// TIA Portal project "Hgu_controller" (V17)

(* hardware
DEVICE "S7-1500/ET200MP station_1"  S7-1500 station
   slot 0: "Rail_0"  Rack  6ES7 590-1***0-0AA0
   slot 1: "HGU_Controller"  CPU 1511-1 PN  6ES7 511-1AK02-0AB0  V2.9
      slot 3: "CPU display_1"  6ES7591-1AA00-0AA0
      slot 32768: "PROFINET interface_1"  X1
         slot 32769: "Port_1"  X1 P1
         slot 32770: "Port_2"  X1 P2
      slot 34817: "Virtual CP interface port_1"  Virtual CP interface port  Virtual CP interface port
DEVICE "ET 200SP station_1"  ET 200SP-Station
   slot 0: "Rack_0"  Rack  6ES5 710-8MAx1
   slot 0: "HPU"  IM 155-6 PN ST  6ES7 155-6AU01-0BN0  V4.2
   slot 1: "DI 16x24VDC ST_1"  DI 16x24VDC ST  6ES7 131-6BH01-0BA0  V0.0
      slot 1: "DI 16x24VDC ST_1"  DI 16x24VDC ST
   slot 2: "DI 16x24VDC ST_2"  DI 16x24VDC ST  6ES7 131-6BH01-0BA0  V0.0
      slot 1: "DI 16x24VDC ST_2"  DI 16x24VDC ST
   slot 3: "DQ 16x24VDC/0.5A ST_1"  DQ 16x24VDC/0.5A ST  6ES7 132-6BH01-0BA0  V0.0
      slot 1: "DQ 16x24VDC/0.5A ST_1"  DQ 16x24VDC/0.5A ST
   slot 4: "AI 4xU/I 2-wire ST_1"  AI 4xU/I 2-wire ST  6ES7 134-6HD01-0BA1  V2.0
      slot 1: "AI 4xU/I 2-wire ST_1"  AI 4xU/I 2-wire ST
   slot 5: "AI 4xU/I 2-wire ST_2"  AI 4xU/I 2-wire ST  6ES7 134-6HD01-0BA1  V2.0
      slot 1: "AI 4xU/I 2-wire ST_2"  AI 4xU/I 2-wire ST
   slot 6: "AI 4xU/I 2-wire ST_3"  AI 4xU/I 2-wire ST  6ES7 134-6HD01-0BA1  V2.0
      slot 1: "AI 4xU/I 2-wire ST_3"  AI 4xU/I 2-wire ST
   slot 7: "AI 4xU/I 2-wire ST_4"  AI 4xU/I 2-wire ST  6ES7 134-6HD01-0BA1  V2.0
      slot 1: "AI 4xU/I 2-wire ST_4"  AI 4xU/I 2-wire ST
   slot 8: "AI 4xU/I 2-wire ST_5"  AI 4xU/I 2-wire ST  6ES7 134-6HD01-0BA1  V2.0
      slot 1: "AI 4xU/I 2-wire ST_5"  AI 4xU/I 2-wire ST
   slot 9: "CM PtP_1"  CM PtP  6ES7 137-6AA00-0BA0  V1.0
      slot 1: "CM PtP_1"  CM PtP Sub
   slot 10: "Server module_1"  Server module  6ES7 193-6PA00-0AA0  V1.1
      slot 1: "Server module_1"  Server module
   slot 127: "BA 2xRJ45"  BA 2xRJ45  6ES7 193-6AR00-0AA0  V0.0
      slot 1: "Port_1"  X1 P1 R  6ES7 193-6AR00-0AA0  V0.0
      slot 2: "Port_2"  X1 P2 R  6ES7 193-6AR00-0AA0  V0.0
DEVICE "SINAMICS G_1"  Sinamics.Device
   slot 0: "	_0"  Rail  SinamicsG120CRackP
   slot 0: "Drive_1"  G120C PN  6SL3210-1KE31-7AF1  4.7.13
      slot 1: "PROFINET interface"  MDD-SinamicsG120-P
      slot 3: "PM G120C"  PM G120C  6SL3210-1KE31-7AF1  -
DEVICE "SINAMICS G_2"  Sinamics.Device
   slot 0: "	_0"  Rail  SinamicsG120CRackP
   slot 0: "Drive_2"  G120C PN  6SL3210-1KE31-7AF1  4.7.13
      slot 1: "PROFINET interface"  MDD-SinamicsG120-P
      slot 3: "PM G120C"  PM G120C  6SL3210-1KE31-7AF1  -
DEVICE "SINAMICS G_3"  Sinamics.Device
   slot 0: "	_0"  Rail  SinamicsG120CRackP
   slot 0: "Drive_3"  G120C PN  6SL3210-1KE31-7AF1  4.7.13
      slot 1: "PROFINET interface"  MDD-SinamicsG120-P
      slot 3: "PM G120C"  PM G120C  6SL3210-1KE31-7AF1  -
DEVICE "SINAMICS G_4"  Sinamics.Device
   slot 0: "	_0"  Rail  SinamicsG120CRackP
   slot 0: "Drive_4"  G120C PN  6SL3210-1KE31-7AF1  4.7.13
      slot 1: "PROFINET interface"  MDD-SinamicsG120-P
      slot 3: "PM G120C"  PM G120C  6SL3210-1KE31-7AF1  -
DEVICE "SINAMICS G_6"  Sinamics.Device
   slot 0: "	_0"  Rail  SinamicsG120CRackP
   slot 0: "Drive_6"  G120C PN  6SL3210-1KE31-7AF1  4.7.13
      slot 1: "PROFINET interface"  MDD-SinamicsG120-P
      slot 3: "PM G120C"  PM G120C  6SL3210-1KE31-7AF1  -
DEVICE "ET 200SP station_2"  ET 200SP-Station
   slot 0: "Rack_0"  Rack  6ES5 710-8MAx1
   slot 0: "Main Cabinet"  IM 155-6 PN ST  6ES7 155-6AU01-0BN0  V4.2
   slot 1: "DI 16x24VDC ST_1"  DI 16x24VDC ST  6ES7 131-6BH01-0BA0  V0.0
      slot 1: "DI 16x24VDC ST_1"  DI 16x24VDC ST
   slot 2: "DI 16x24VDC ST_2"  DI 16x24VDC ST  6ES7 131-6BH01-0BA0  V0.0
      slot 1: "DI 16x24VDC ST_2"  DI 16x24VDC ST
   slot 3: "DQ 16x24VDC/0.5A ST_1"  DQ 16x24VDC/0.5A ST  6ES7 132-6BH01-0BA0  V0.0
      slot 1: "DQ 16x24VDC/0.5A ST_1"  DQ 16x24VDC/0.5A ST
   slot 4: "Server module_01"  Server module  6ES7 193-6PA00-0AA0  V1.1
      slot 1: "Server module_01"  Server module
   slot 127: "BA 2xRJ45"  BA 2xRJ45  6ES7 193-6AR00-0AA0  V0.0
      slot 1: "Port_1"  X1 P1 R  6ES7 193-6AR00-0AA0  V0.0
      slot 2: "Port_2"  X1 P2 R  6ES7 193-6AR00-0AA0  V0.0
*)

// ===== PLC "HGU_Controller"  CPU 1511-1 PN =====

VAR_GLOBAL   // PLC tag table "Default tag table"
   "Motor1MpcbFault" AT %I44.0 : Bool;   // Motor1 Mks Termik Hata
   "Motor2MpcbFault" AT %I44.1 : Bool;   // Motor 2 Mks Termik Hata
   "Motor3MpcbFault" AT %I44.2 : Bool;   // Motor 3 Mks Termik Hata
   "Motor4MpcbFault" AT %I44.3 : Bool;   // Motor 4 Mks Termik Hata
   "Motor5MpcbFault" AT %I44.4 : Bool;   // Motor 5 Mks Termik Hata
   "Motor6MpcbFault" AT %I44.5 : Bool;   // Motor 6 Mks Termik Hata
   "CoilTubeSoftStarterRunning" AT %I44.6 : Bool;   // Coiltube Yumuşak Yol Verici Çalışıyor
   "CoilTubeSoftStarterContactor" AT %I44.7 : Bool;   // Coiltube Yumuşak Yol Verici Kontaktör Devrede
   "CoilTubeMpcbFault" AT %I45.0 : Bool;   // Coiltube Mks Termik Hata
   "CircSoftStarterRunning" AT %I45.1 : Bool;   // Sirkülasyon Yumuşak Yol Verici Çalışıyor
   "CircSoftStarterContactor" AT %I45.2 : Bool;   // Sirkülasyon Yumuşak Yol Verici Kontaktör Devrede
   "CircMpcbFault" AT %I45.3 : Bool;   // Sirkülasyon Mks Termik Hata
   "ParticleContactorEngaged" AT %I45.4 : Bool;   // Particle Measurement Contactor Engaged
   "ParticleMpcbFault" AT %I45.5 : Bool;   // Particle Measurement Mks Termik Hata
   "PhaseProtectionOk" AT %I45.6 : Bool;   // Faz Koruma Rölesi Ok
   "SafetyRelayOk" AT %I45.7 : Bool;   // Emniyet Rölesi Ok
   "MainSwitchAlarm" AT %I46.0 : Bool;   // Ana Şalter Alarm Kontağı
   "ToroidalLeakageFuse" AT %I46.1 : Bool;   // Toroidal Kaçak Akım Rölesi Sigorta Bilgisi
   "ToroidalLeakageAlarm" AT %I46.2 : Bool;   // Toroidal Kaçak Akım Rölesi Alarm
   "EmergencyStopPlcStatus" AT %I46.3 : Bool;   // Acil Stop Butonu Plc Durum
   "EmergencyStopGpStatus" AT %I46.4 : Bool;   // Acil Stop Butonu Gb Durum
   "ControlPhaseFuse220Vac" AT %I46.5 : Bool;   // 220Vac Kumanda Faz Sigortası Bilgisi
   "EnergyAnalyzerLeakageRelay" AT %I46.6 : Bool;   // Enerji Analizörü Besleme Kaçak Akım Rölesi
   "SignalTowerGreen" AT %Q20.0 : Bool;   // Işık Kulesi Yeşil
   "SignalTowerYellow" AT %Q20.1 : Bool;   // Işık Kulesi Sarı
   "SignalTowerRed" AT %Q20.2 : Bool;   // Işık Kulesi Kırmızı
   "SignalTowerBuzzer" AT %Q20.3 : Bool;   // Işık Kulesi Buzzer
   "ParticleMotorCmd" AT %Q20.4 : Bool;   // Particle Measurement Motor 1/0 Komutu
   "CircContactorCmd" AT %Q20.5 : Bool;   // Sirkülasyon Kontaktör Komutu
   "CircSoftStarterCmd" AT %Q20.6 : Bool;   // Sirkülasyon Yumuşak Yol Verici Komutu
   "CoilTubeContactorCmd" AT %Q20.7 : Bool;   // Coiltube Kontaktör Komutu
   "CoilTubeSoftStarterCmd" AT %Q21.0 : Bool;   // Coiltube Yumuşak Yol Verici Komutu
   "EmergencyStopUnit1" AT %I0.0 : Bool;   // Acil Durdurma Butonu Ünite 1
   "EmergencyStopUnit2" AT %I0.1 : Bool;   // Acil Durdurma Butonu Ünite 2
   "EmergencyStopUnit3" AT %I0.2 : Bool;   // Acil Durdurma Butonu Ünite 3
   "EmergencyStopUnit4" AT %I0.3 : Bool;   // Acil Durdurma Butonu Ünite 4
   "Motor1FilterWarning" AT %I0.4 : Bool;   // Motor 1 Basınç Hattı Filtresi Uyarı
   "Motor1FilterError" AT %I0.5 : Bool;   // Motor 1 Basınç Hattı Filtresi Hata
   "Motor2FilterWarning" AT %I0.6 : Bool;   // Motor 2 Basınç Hattı Filtresi Uyarı
   "Motor2FilterError" AT %I0.7 : Bool;   // Motor 2 Basınç Hattı Filtresi Hata
   "Motor3FilterWarning" AT %I1.0 : Bool;   // Motor 3 Basınç Hattı Filtresi Uyarı
   "Motor3FilterError" AT %I1.1 : Bool;   // Motor 3 Basınç Hattı Filtresi Hata
   "Motor4FilterWarning" AT %I1.2 : Bool;   // Motor 4 Basınç Hattı Filtresi Uyarı
   "Motor4FilterError" AT %I1.3 : Bool;   // Motor 4 Basınç Hattı Filtresi Hata
   "Motor5FilterWarning" AT %I1.4 : Bool;   // Motor 5 Basınç Hattı Filtresi Uyarı
   "Motor5FilterError" AT %I1.5 : Bool;   // Motor 5 Basınç Hattı Filtresi Hata
   "Motor6FilterWarning" AT %I1.6 : Bool;   // Motor 6 Basınç Hattı Filtresi Uyarı
   "Motor6FilterError" AT %I1.7 : Bool;   // Motor 6 Basınç Hattı Filtresi Hata
   "CoilTubeFilterWarning" AT %I2.0 : Bool;   // Coiltube Basınç Hattı Filtresi Uyarı
   "CoilTubeFilterError" AT %I2.1 : Bool;   // Coiltube Basınç Hattı Filtresi Hata
   "TankMinLevelSwitch" AT %I2.2 : Bool;   // Tank Min Seviye Şalteri
   "TankMaxLevelSwitch" AT %I2.3 : Bool;   // Tank Max Seviye Şalteri
   "Motor1CompensatedValve" AT %I2.4 : Bool;   // Motor 1 Kompansatörlü Vana
   "Motor2CompensatedValve" AT %I2.5 : Bool;   // Motor 2 Kompansatörlü Vana
   "Motor3CompensatedValve" AT %I2.6 : Bool;   // Motor 3 Kompansatörlü Vana
   "Motor4CompensatedValve" AT %I2.7 : Bool;   // Motor 4 Kompansatörlü Vana
   "Motor5CompensatedValve" AT %I3.0 : Bool;   // Motor 5 Kompansatörlü Vana
   "Motor6CompensatedValve" AT %I3.1 : Bool;   // Motor 6 Kompansatörlü Vana
   "ChillerWaterFlowSensor" AT %I3.2 : Bool;   // Chiller Su Akış Sensoru
   "TemperatureSensor" AT %IW4 : Int;   // Sıcaklık Sensörü
   "ContinuousLevelSensor" AT %IW6 : Int;   // Sürekli Seviye Sensörü
   "AquaSensor" AT %IW8 : Int;   // Aqua Sensörü
   "PressureTransmitter1" AT %IW10 : Int;   // Basınç Transmitteri 1
   "PressureTransmitter2" AT %IW12 : Int;   // Basınç Transmitteri 2
   "PressureTransmitter3" AT %IW14 : Int;   // Basınç Transmitteri 3
   "PressureTransmitter4" AT %IW16 : Int;   // Basınç Transmitteri 4
   "PressureTransmitter5" AT %IW18 : Int;   // Basınç Transmitteri 5
   "PressureTransmitter6" AT %IW20 : Int;   // Basınç Transmitteri 6
   "CoilTubePressureTransmitter" AT %IW22 : Int;   // Coiltube Basınç Transmitteri
   "Hsm1PressureTransmitter" AT %IW24 : Int;   // Hsm1 Basınç Transmitteri
   "Hsm2PressureTransmitter" AT %IW26 : Int;   // Hsm2 Basınç Transmitteri
   "Hsm3PressureTransmitter" AT %IW28 : Int;   // Hsm3 Basınç Transmitteri
   "Hsm4PressureTransmitter" AT %IW30 : Int;   // Hsm4 Basınç Transmitteri
   "Hsm5PressureTransmitter" AT %IW32 : Int;   // Hsm5 Basınç Transmitteri
   "Hsm6PressureTransmitter" AT %IW34 : Int;   // Hsm6 Basınç Transmitteri
   "Hsm7PressureTransmitter" AT %IW48 : Int;   // Hsm7 Basınç Transmitteri
   "ChillerInletTemperature" AT %IW50 : Int;   // Chiller Giriş Sıcaklığı
   "ChillerOutletTemperature" AT %IW52 : Int;   // Chiller Çıkış Sıcaklığı
   "M1_Control_Word" AT %QW100 : Int;
   "M1_RPM_Setpoint_Word" AT %QW102 : Int;
   "M1_Reserved_1" AT %QW104 : Int;
   "M1_Reserved_2" AT %QW106 : Int;
   "M1_Reserved_3" AT %QW108 : Int;
   "M1_Reserved_4" AT %QW110 : Int;
   "M1_Status_Word" AT %IW100 : Int;
   "M1_RPM_Actual_Word" AT %IW102 : Int;
   "M1_Current_Word" AT %IW104 : Int;
   "M1_Temperature_Word" AT %IW106 : Int;
   "M1_Error_Word" AT %IW108 : Int;
   "M1_Diagnostic_Word" AT %IW110 : Int;
   "M2_RPM_Setpoint_Word" AT %QW122 : Int;
   "M2_Reserved_1" AT %QW124 : Int;
   "M2_Reserved_2" AT %QW126 : Int;
   "M2_Reserved_3" AT %QW128 : Int;
   "M2_Reserved_4" AT %QW130 : Int;
   "M2_Status_Word" AT %IW120 : Int;
   "M2_RPM_Actual_Word" AT %IW122 : Int;
   "M2_Current_Word" AT %IW124 : Int;
   "M2_Temperature_Word" AT %IW126 : Int;
   "M2_Error_Word" AT %IW128 : Int;
   "M2_Diagnostic_Word" AT %IW130 : Int;
   "M3_Control_Word" AT %QW140 : Int;
   "M3_RPM_Setpoint_Word" AT %QW142 : Int;
   "M3_Reserved_1" AT %QW144 : Int;
   "M3_Reserved_2" AT %QW146 : Int;
   "M3_Reserved_3" AT %QW148 : Int;
   "M3_Reserved_4" AT %QW150 : Int;
   "M3_Status_Word" AT %IW140 : Int;
   "M3_RPM_Actual_Word" AT %IW142 : Int;
   "M3_Current_Word" AT %IW144 : Int;
   "M3_Temperature_Word" AT %IW146 : Int;
   "M3_Error_Word" AT %IW148 : Int;
   "M3_Diagnostic_Word" AT %IW150 : Int;
   "M4_Control_Word" AT %QW160 : Int;
   "M4_RPM_Setpoint_Word" AT %QW162 : Int;
   "M4_Reserved_1" AT %QW164 : Int;
   "M4_Reserved_2" AT %QW166 : Int;
   "M4_Reserved_3" AT %QW168 : Int;
   "M4_Reserved_4" AT %QW170 : Int;
   "M4_Status_Word" AT %IW160 : Int;
   "M4_RPM_Actual_Word" AT %IW162 : Int;
   "M4_Current_Word" AT %IW164 : Int;
   "M4_Temperature_Word" AT %IW166 : Int;
   "M4_Error_Word" AT %IW168 : Int;
   "M4_Diagnostic_Word" AT %IW170 : Int;
   "M5_Control_Word" AT %QW180 : Int;
   "M5_RPM_Setpoint_Word" AT %QW182 : Int;
   "M5_Reserved_1" AT %QW184 : Int;
   "M5_Reserved_2" AT %QW186 : Int;
   "M5_Reserved_3" AT %QW188 : Int;
   "M5_Reserved_4" AT %QW190 : Int;
   "M5_Status_Word" AT %IW180 : Int;
   "M5_RPM_Actual_Word" AT %IW182 : Int;
   "M5_Current_Word" AT %IW184 : Int;
   "M5_Temperature_Word" AT %IW186 : Int;
   "M5_Error_Word" AT %IW188 : Int;
   "M5_Diagnostic_Word" AT %IW190 : Int;
   "M6_Control_Word" AT %QW200 : Int;
   "M6_RPM_Setpoint_Word" AT %QW202 : Int;
   "M6_Reserved_1" AT %QW204 : Int;
   "M6_Reserved_2" AT %QW206 : Int;
   "M6_Reserved_3" AT %QW208 : Int;
   "M6_Reserved_4" AT %QW210 : Int;
   "M6_Status_Word" AT %IW200 : Int;
   "M6_RPM_Actual_Word" AT %IW202 : Int;
   "M6_Current_Word" AT %IW204 : Int;
   "M6_Temperature_Word" AT %IW206 : Int;
   "M6_Error_Word" AT %IW208 : Int;
   "M6_Diagnostic_Word" AT %IW210 : Int;
   "M2_Control_Word" AT %IW112 : Int;
END_VAR

DATA_BLOCK "DB_HGU_Execution_V17"   // DB1
TITLE = 'HGU Execution Variables Data Block - V17 PUMP Naming Convention'
{ S7_Optimized_Access := 'TRUE' }
VERSION : 3.0
// =============================================================================
//  TUSAÅž HGU CONTROL SYSTEM - EXECUTION VARIABLES DATA BLOCK V17
//  TIA Portal S7-1500 Structured Control Language (SCL)
//  Updated: 2025-08-15 - V17 PUMP NAMING CONVENTION
//  Description: All execution variables with PUMP/MOTOR/VALVE naming clarity
//  =============================================================================
//  =============================================================================
//  SYSTEM CONTROL AND STATUS - INTEGRATED ARCHITECTURE
//  =============================================================================
   VAR
      SYSTEM_ENABLE : Bool := FALSE;   // Master system enable
      SYSTEM_READY : Bool := FALSE;   // All subsystems ready
      SYSTEM_ERROR : Bool := FALSE;   // Any system error active
      EMERGENCY_STOP : Bool := FALSE;   // Emergency stop status
      RESET_ERRORS : Bool := FALSE;   // Reset all errors command
      DEBUG_MODE : Bool := FALSE;   // Debug mode enable System Performance Monitoring
      SYSTEM_CYCLE_COUNTER : UDInt := 0;   // System cycle counter
      SYSTEM_SCAN_TIME : UDInt := 0;   // Current scan time (ms)
      LAST_UPDATE_TIME : DTL;   // Last system update time ============================================================================= SYSTEM SETPOINTS AND TOTALS =============================================================================
      SYSTEM_PRESSURE_SETPOINT : Real := 280.0;   // System pressure setpoint (bar) - UI adjustable
      SYSTEM_FLOW_SETPOINT : Real := 180.0;   // System flow setpoint (L/min) - UI adjustable
      TOTAL_SYSTEM_FLOW : Real := 0.0;   // Total system flow rate (L/min)
      TOTAL_SYSTEM_PRESSURE : Real := 0.0;   // Average system pressure (bar)
      ACTIVE_MOTOR_COUNT : USInt := 0;   // Currently active motors
      SYSTEM_EFFICIENCY : Real := 0.0;   // Overall system efficiency (%)
      SYSTEM_STATUS : Int := 0;   // System status (0=Init, 1=Ready, 2=Running, 3=Error)
      SYSTEM_SAFETY_STATUS : Int := 0;   // Safety status (0=Unknown, 1=Safe, 2=Safety Error)
      SYSTEM_PRESSURE_AVERAGE : Real := 0.0;   // System pressure average (bar)
      SYSTEM_ACTIVE_PUMPS : Int := 0;   // Active pumps count ============================================================================= PUMP #1 VARIABLES (Pressure & Flow Control) =============================================================================
      PUMP_1_PRESSURE_SETPOINT : Real := 280.0;   // Pump 1 Pressure Setpoint (Bar) - Load Sensing coordinated
      PUMP_1_PRESSURE_ACTUAL : Real := 0.0;   // Pump 1 Actual Pressure (Bar) - Sensor feedback
      PUMP_1_FLOW_SETPOINT : Real := 30.0;   // Pump 1 Flow Setpoint (L/min) - User adjustable
      PUMP_1_FLOW_ACTUAL : Real := 0.0;   // Pump 1 Actual Flow (L/min) - Calculated value
      PUMP_1_LEAK_RATE : Real := 0.0;   // Pump 1 Leak Rate (L/min) - Diagnostic value
      PUMP_1_ENABLED : Bool := FALSE;   // Pump 1 Enable Control (PID enable) ============================================================================= MOTOR #1 VARIABLES (Electrical Parameters) =============================================================================
      MOTOR_1_RPM_SETPOINT : Real := 1000.0;   // Motor 1 Target RPM - VFD setpoint
      MOTOR_1_RPM_ACTUAL : Real := 0.0;   // Motor 1 Actual RPM - Encoder feedback
      MOTOR_1_CURRENT_A : Real := 0.0;   // Motor 1 Current (A) - Electrical measurement
      MOTOR_1_TEMPERATURE_C : Real := 25.0;   // Motor 1 Temperature (Â°C) - Thermal monitoring
      MOTOR_1_ENABLE : Bool := FALSE;   // Motor 1 Enable Control
      MOTOR_1_STATUS : USInt := 0;   // Motor 1 Status (0=Offline, 1=Ready, 2=Running, 3=Error)
      MOTOR_1_ERROR_CODE : USInt := 0;   // Motor 1 Error code - Diagnostic information
      MOTOR_1_START_CMD : Bool := FALSE;   // Motor 1 Start Command
      MOTOR_1_STOP_CMD : Bool := FALSE;   // Motor 1 Stop Command
      MOTOR_1_RESET_CMD : Bool := FALSE;   // Motor 1 Reset Command
      MOTOR_1_START_ACK : Bool := FALSE;   // Motor 1 Start Acknowledgment
      MOTOR_1_STOP_ACK : Bool := FALSE;   // Motor 1 Stop Acknowledgment
      MOTOR_1_RESET_ACK : Bool := FALSE;   // Motor 1 Reset Acknowledgment G120C FREE Telegram Variables - REMOVED Physical I/O mapping done via TAG Table (M1_Control_Word, M1_Status_Word, etc.) ============================================================================= VALVE #1 VARIABLES (Position Control) =============================================================================
      VALVE_1_CURRENT_SETPOINT : Real := 0.0;   // Valve 1 Current Setpoint (0-10000) - Control output
      VALVE_1_CURRENT_MA : Real := 4.0;   // Valve 1 Current (4-20mA) - Analog signal
      PUMP_1_LINE_FILTER_STATUS : USInt := 2;   // Pump 1 Line Filter - Pompa Ã§Ä±kÄ±ÅŸÄ±nda (0=Error, 1=Warning, 2=OK)
      PUMP_1_SUCTION_FILTER_STATUS : USInt := 1;   // Pump 1 Suction Filter - Pompa giriÅŸinde (0=Error, 1=OK)
      PUMP_1_MANUAL_VALVE_STATUS : USInt := 1;   // Pump 1 Manual Valve - Tank-Pompa arasÄ± (0=KapalÄ±, 1=AÃ§Ä±k) ============================================================================= PUMP #2 VARIABLES (Pressure & Flow Control) =============================================================================
      PUMP_2_PRESSURE_SETPOINT : Real := 280.0;   // Pump 2 Pressure Setpoint (Bar) - Load Sensing coordinated
      PUMP_2_PRESSURE_ACTUAL : Real := 0.0;   // Pump 2 Actual Pressure (Bar) - Sensor feedback
      PUMP_2_FLOW_SETPOINT : Real := 30.0;   // Pump 2 Flow Setpoint (L/min) - User adjustable
      PUMP_2_FLOW_ACTUAL : Real := 0.0;   // Pump 2 Actual Flow (L/min) - Calculated value
      PUMP_2_LEAK_RATE : Real := 0.0;   // Pump 2 Leak Rate (L/min) - Diagnostic value
      PUMP_2_ENABLED : Bool := FALSE;   // Pump 2 Enable Control (PID enable) ============================================================================= MOTOR #2 VARIABLES (Electrical Parameters) =============================================================================
      MOTOR_2_RPM_SETPOINT : Real := 1000.0;   // Motor 2 Target RPM - VFD setpoint
      MOTOR_2_RPM_ACTUAL : Real := 0.0;   // Motor 2 Actual RPM - Encoder feedback
      MOTOR_2_CURRENT_A : Real := 0.0;   // Motor 2 Current (A) - Electrical measurement
      MOTOR_2_TEMPERATURE_C : Real := 25.0;   // Motor 2 Temperature (Â°C) - Thermal monitoring
      MOTOR_2_ENABLE : Bool := FALSE;   // Motor 2 Enable Control
      MOTOR_2_STATUS : USInt := 0;   // Motor 2 Status (0=Offline, 1=Ready, 2=Running, 3=Error)
      MOTOR_2_ERROR_CODE : USInt := 0;   // Motor 2 Error code - Diagnostic information
      MOTOR_2_START_CMD : Bool := FALSE;   // Motor 2 Start Command
      MOTOR_2_STOP_CMD : Bool := FALSE;   // Motor 2 Stop Command
      MOTOR_2_RESET_CMD : Bool := FALSE;   // Motor 2 Reset Command
      MOTOR_2_START_ACK : Bool := FALSE;   // Motor 2 Start Acknowledgment
      MOTOR_2_STOP_ACK : Bool := FALSE;   // Motor 2 Stop Acknowledgment
      MOTOR_2_RESET_ACK : Bool := FALSE;   // Motor 2 Reset Acknowledgment G120C FREE Telegram Variables - REMOVED (Use M2_* TAGs) ============================================================================= VALVE #2 VARIABLES (Position Control) =============================================================================
      VALVE_2_CURRENT_SETPOINT : Real := 0.0;   // Valve 2 Current Setpoint (0-10000) - Control output
      VALVE_2_CURRENT_MA : Real := 4.0;   // Valve 2 Current (4-20mA) - Analog signal
      PUMP_2_LINE_FILTER_STATUS : USInt := 2;   // Pump 2 Line Filter - Pompa Ã§Ä±kÄ±ÅŸÄ±nda (0=Error, 1=Warning, 2=OK)
      PUMP_2_SUCTION_FILTER_STATUS : USInt := 1;   // Pump 2 Suction Filter - Pompa giriÅŸinde (0=Error, 1=OK)
      PUMP_2_MANUAL_VALVE_STATUS : USInt := 1;   // Pump 2 Manual Valve - Tank-Pompa arasÄ± (0=KapalÄ±, 1=AÃ§Ä±k) ============================================================================= PUMP #3 VARIABLES (Pressure & Flow Control) =============================================================================
      PUMP_3_PRESSURE_SETPOINT : Real := 280.0;   // Pump 3 Pressure Setpoint (Bar) - Load Sensing coordinated
      PUMP_3_PRESSURE_ACTUAL : Real := 0.0;   // Pump 3 Actual Pressure (Bar) - Sensor feedback
      PUMP_3_FLOW_SETPOINT : Real := 30.0;   // Pump 3 Flow Setpoint (L/min) - User adjustable
      PUMP_3_FLOW_ACTUAL : Real := 0.0;   // Pump 3 Actual Flow (L/min) - Calculated value
      PUMP_3_LEAK_RATE : Real := 0.0;   // Pump 3 Leak Rate (L/min) - Diagnostic value
      PUMP_3_ENABLED : Bool := FALSE;   // Pump 3 Enable Control (PID enable) ============================================================================= MOTOR #3 VARIABLES (Electrical Parameters) =============================================================================
      MOTOR_3_RPM_SETPOINT : Real := 1000.0;   // Motor 3 Target RPM - VFD setpoint
      MOTOR_3_RPM_ACTUAL : Real := 0.0;   // Motor 3 Actual RPM - Encoder feedback
      MOTOR_3_CURRENT_A : Real := 0.0;   // Motor 3 Current (A) - Electrical measurement
      MOTOR_3_TEMPERATURE_C : Real := 25.0;   // Motor 3 Temperature (Â°C) - Thermal monitoring
      MOTOR_3_ENABLE : Bool := FALSE;   // Motor 3 Enable Control
      MOTOR_3_STATUS : USInt := 0;   // Motor 3 Status (0=Offline, 1=Ready, 2=Running, 3=Error)
      MOTOR_3_ERROR_CODE : USInt := 0;   // Motor 3 Error code - Diagnostic information
      MOTOR_3_START_CMD : Bool := FALSE;   // Motor 3 Start Command
      MOTOR_3_STOP_CMD : Bool := FALSE;   // Motor 3 Stop Command
      MOTOR_3_RESET_CMD : Bool := FALSE;   // Motor 3 Reset Command
      MOTOR_3_START_ACK : Bool := FALSE;   // Motor 3 Start Acknowledgment
      MOTOR_3_STOP_ACK : Bool := FALSE;   // Motor 3 Stop Acknowledgment
      MOTOR_3_RESET_ACK : Bool := FALSE;   // Motor 3 Reset Acknowledgment G120C FREE Telegram Variables - REMOVED (Use M5)
      MOTOR_3_CONTROL_WORD : Word;   // 140 : Word; // Motor 3 Control Word (PZD[0] Send)
      MOTOR_3_RPM_SETPOINT_WORD : Int;   // 142 : Int; // Motor 3 RPM Setpoint Word (PZD[1] Send)
      MOTOR_3_RESERVED_1 : Word;   // 144 : Word; // Motor 3 Reserved PZD[2] Send
      MOTOR_3_RESERVED_2 : Word;   // 146 : Word; // Motor 3 Reserved PZD[3] Send
      MOTOR_3_RESERVED_3 : Word;   // 148 : Word; // Motor 3 Reserved PZD[4] Send
      MOTOR_3_RESERVED_4 : Word;   // 150 : Word; // Motor 3 Reserved PZD[5] Send
      MOTOR_3_STATUS_WORD : Word;   // 140 : Word; // Motor 3 Status Word (PZD[0] Receive)
      MOTOR_3_RPM_ACTUAL_WORD : Int;   // 142 : Int; // Motor 3 RPM Actual Word (PZD[1] Receive)
      MOTOR_3_CURRENT_WORD : Int;   // 144 : Int; // Motor 3 Current Word (PZD[2] Receive)
      MOTOR_3_TEMPERATURE_WORD : Int;   // 146 : Int; // Motor 3 Temperature Word (PZD[3] Receive)
      MOTOR_3_ERROR_WORD : Word;   // 148 : Word; // Motor 3 Error/Warning Word (PZD[4] Receive)
      MOTOR_3_DIAGNOSTIC_WORD : Word;   // 150 : Word; // Motor 3 Diagnostic Word (PZD[5] Receive) ============================================================================= VALVE #3 VARIABLES (Position Control) =============================================================================
      VALVE_3_CURRENT_SETPOINT : Real := 0.0;   // Valve 3 Current Setpoint (0-10000) - Control output
      VALVE_3_CURRENT_MA : Real := 4.0;   // Valve 3 Current (4-20mA) - Analog signal
      PUMP_3_LINE_FILTER_STATUS : USInt := 2;   // Pump 3 Line Filter - Pompa Ã§Ä±kÄ±ÅŸÄ±nda (0=Error, 1=Warning, 2=OK)
      PUMP_3_SUCTION_FILTER_STATUS : USInt := 1;   // Pump 3 Suction Filter - Pompa giriÅŸinde (0=Error, 1=OK)
      PUMP_3_MANUAL_VALVE_STATUS : USInt := 1;   // Pump 3 Manual Valve - Tank-Pompa arasÄ± (0=KapalÄ±, 1=AÃ§Ä±k) ============================================================================= PUMP #4 VARIABLES (Pressure & Flow Control) =============================================================================
      PUMP_4_PRESSURE_SETPOINT : Real := 280.0;   // Pump 4 Pressure Setpoint (Bar) - Load Sensing coordinated
      PUMP_4_PRESSURE_ACTUAL : Real := 0.0;   // Pump 4 Actual Pressure (Bar) - Sensor feedback
      PUMP_4_FLOW_SETPOINT : Real := 30.0;   // Pump 4 Flow Setpoint (L/min) - User adjustable
      PUMP_4_FLOW_ACTUAL : Real := 0.0;   // Pump 4 Actual Flow (L/min) - Calculated value
      PUMP_4_LEAK_RATE : Real := 0.0;   // Pump 4 Leak Rate (L/min) - Diagnostic value
      PUMP_4_ENABLED : Bool := FALSE;   // Pump 4 Enable Control (PID enable) ============================================================================= MOTOR #4 VARIABLES (Electrical Parameters) =============================================================================
      MOTOR_4_RPM_SETPOINT : Real := 1000.0;   // Motor 4 Target RPM - VFD setpoint
      MOTOR_4_RPM_ACTUAL : Real := 0.0;   // Motor 4 Actual RPM - Encoder feedback
      MOTOR_4_CURRENT_A : Real := 0.0;   // Motor 4 Current (A) - Electrical measurement
      MOTOR_4_TEMPERATURE_C : Real := 25.0;   // Motor 4 Temperature (Â°C) - Thermal monitoring
      MOTOR_4_ENABLE : Bool := FALSE;   // Motor 4 Enable Control
      MOTOR_4_STATUS : USInt := 0;   // Motor 4 Status (0=Offline, 1=Ready, 2=Running, 3=Error)
      MOTOR_4_ERROR_CODE : USInt := 0;   // Motor 4 Error code - Diagnostic information
      MOTOR_4_START_CMD : Bool := FALSE;   // Motor 4 Start Command
      MOTOR_4_STOP_CMD : Bool := FALSE;   // Motor 4 Stop Command
      MOTOR_4_RESET_CMD : Bool := FALSE;   // Motor 4 Reset Command
      MOTOR_4_START_ACK : Bool := FALSE;   // Motor 4 Start Acknowledgment
      MOTOR_4_STOP_ACK : Bool := FALSE;   // Motor 4 Stop Acknowledgment
      MOTOR_4_RESET_ACK : Bool := FALSE;   // Motor 4 Reset Acknowledgment G120C FREE Telegram Variables - REMOVED (Use M6)
      MOTOR_4_CONTROL_WORD : Word;   // 160 : Word; // Motor 4 Control Word (PZD[0] Send)
      MOTOR_4_RPM_SETPOINT_WORD : Int;   // 162 : Int; // Motor 4 RPM Setpoint Word (PZD[1] Send)
      MOTOR_4_RESERVED_1 : Word;   // 164 : Word; // Motor 4 Reserved PZD[2] Send
      MOTOR_4_RESERVED_2 : Word;   // 166 : Word; // Motor 4 Reserved PZD[3] Send
      MOTOR_4_RESERVED_3 : Word;   // 168 : Word; // Motor 4 Reserved PZD[4] Send
      MOTOR_4_RESERVED_4 : Word;   // 170 : Word; // Motor 4 Reserved PZD[5] Send
      MOTOR_4_STATUS_WORD : Word;   // 160 : Word; // Motor 4 Status Word (PZD[0] Receive)
      MOTOR_4_RPM_ACTUAL_WORD : Int;   // 162 : Int; // Motor 4 RPM Actual Word (PZD[1] Receive)
      MOTOR_4_CURRENT_WORD : Int;   // 164 : Int; // Motor 4 Current Word (PZD[2] Receive)
      MOTOR_4_TEMPERATURE_WORD : Int;   // 166 : Int; // Motor 4 Temperature Word (PZD[3] Receive)
      MOTOR_4_ERROR_WORD : Word;   // 168 : Word; // Motor 4 Error/Warning Word (PZD[4] Receive)
      MOTOR_4_DIAGNOSTIC_WORD : Word;   // 170 : Word; // Motor 4 Diagnostic Word (PZD[5] Receive) ============================================================================= VALVE #4 VARIABLES (Position Control) =============================================================================
      VALVE_4_CURRENT_SETPOINT : Real := 0.0;   // Valve 4 Current Setpoint (0-10000) - Control output
      VALVE_4_CURRENT_MA : Real := 4.0;   // Valve 4 Current (4-20mA) - Analog signal
      PUMP_4_LINE_FILTER_STATUS : USInt := 2;   // Pump 4 Line Filter - Pompa Ã§Ä±kÄ±ÅŸÄ±nda (0=Error, 1=Warning, 2=OK)
      PUMP_4_SUCTION_FILTER_STATUS : USInt := 1;   // Pump 4 Suction Filter - Pompa giriÅŸinde (0=Error, 1=OK)
      PUMP_4_MANUAL_VALVE_STATUS : USInt := 1;   // Pump 4 Manual Valve - Tank-Pompa arasÄ± (0=KapalÄ±, 1=AÃ§Ä±k) ============================================================================= PUMP #5 VARIABLES (Pressure & Flow Control) =============================================================================
      PUMP_5_PRESSURE_SETPOINT : Real := 280.0;   // Pump 5 Pressure Setpoint (Bar) - Load Sensing coordinated
      PUMP_5_PRESSURE_ACTUAL : Real := 0.0;   // Pump 5 Actual Pressure (Bar) - Sensor feedback
      PUMP_5_FLOW_SETPOINT : Real := 30.0;   // Pump 5 Flow Setpoint (L/min) - User adjustable
      PUMP_5_FLOW_ACTUAL : Real := 0.0;   // Pump 5 Actual Flow (L/min) - Calculated value
      PUMP_5_LEAK_RATE : Real := 0.0;   // Pump 5 Leak Rate (L/min) - Diagnostic value
      PUMP_5_ENABLED : Bool := FALSE;   // Pump 5 Enable Control (PID enable) ============================================================================= MOTOR #5 VARIABLES (Electrical Parameters) =============================================================================
      MOTOR_5_RPM_SETPOINT : Real := 1000.0;   // Motor 5 Target RPM - VFD setpoint
      MOTOR_5_RPM_ACTUAL : Real := 0.0;   // Motor 5 Actual RPM - Encoder feedback
      MOTOR_5_CURRENT_A : Real := 0.0;   // Motor 5 Current (A) - Electrical measurement
      MOTOR_5_TEMPERATURE_C : Real := 25.0;   // Motor 5 Temperature (Â°C) - Thermal monitoring
      MOTOR_5_ENABLE : Bool := FALSE;   // Motor 5 Enable Control
      MOTOR_5_STATUS : USInt := 0;   // Motor 5 Status (0=Offline, 1=Ready, 2=Running, 3=Error)
      MOTOR_5_ERROR_CODE : USInt := 0;   // Motor 5 Error code - Diagnostic information
      MOTOR_5_START_CMD : Bool := FALSE;   // Motor 5 Start Command
      MOTOR_5_STOP_CMD : Bool := FALSE;   // Motor 5 Stop Command
      MOTOR_5_RESET_CMD : Bool := FALSE;   // Motor 5 Reset Command
      MOTOR_5_START_ACK : Bool := FALSE;   // Motor 5 Start Acknowledgment
      MOTOR_5_STOP_ACK : Bool := FALSE;   // Motor 5 Stop Acknowledgment
      MOTOR_5_RESET_ACK : Bool := FALSE;   // Motor 5 Reset Acknowledgment G120C FREE Telegram Variables - REMOVED (Use M7)
      MOTOR_5_CONTROL_WORD : Word;   // 180 : Word; // Motor 5 Control Word (PZD[0] Send)
      MOTOR_5_RPM_SETPOINT_WORD : Int;   // 182 : Int; // Motor 5 RPM Setpoint Word (PZD[1] Send)
      MOTOR_5_RESERVED_1 : Word;   // 184 : Word; // Motor 5 Reserved PZD[2] Send
      MOTOR_5_RESERVED_2 : Word;   // 186 : Word; // Motor 5 Reserved PZD[3] Send
      MOTOR_5_RESERVED_3 : Word;   // 188 : Word; // Motor 5 Reserved PZD[4] Send
      MOTOR_5_RESERVED_4 : Word;   // 190 : Word; // Motor 5 Reserved PZD[5] Send
      MOTOR_5_STATUS_WORD : Word;   // 180 : Word; // Motor 5 Status Word (PZD[0] Receive)
      MOTOR_5_RPM_ACTUAL_WORD : Int;   // 182 : Int; // Motor 5 RPM Actual Word (PZD[1] Receive)
      MOTOR_5_CURRENT_WORD : Int;   // 184 : Int; // Motor 5 Current Word (PZD[2] Receive)
      MOTOR_5_TEMPERATURE_WORD : Int;   // 186 : Int; // Motor 5 Temperature Word (PZD[3] Receive)
      MOTOR_5_ERROR_WORD : Word;   // 188 : Word; // Motor 5 Error/Warning Word (PZD[4] Receive)
      MOTOR_5_DIAGNOSTIC_WORD : Word;   // 190 : Word; // Motor 5 Diagnostic Word (PZD[5] Receive) ============================================================================= VALVE #5 VARIABLES (Position Control) =============================================================================
      VALVE_5_CURRENT_SETPOINT : Real := 0.0;   // Valve 5 Current Setpoint (0-10000) - Control output
      VALVE_5_CURRENT_MA : Real := 4.0;   // Valve 5 Current (4-20mA) - Analog signal
      PUMP_5_LINE_FILTER_STATUS : USInt := 2;   // Pump 5 Line Filter - Pompa Ã§Ä±kÄ±ÅŸÄ±nda (0=Error, 1=Warning, 2=OK)
      PUMP_5_SUCTION_FILTER_STATUS : USInt := 1;   // Pump 5 Suction Filter - Pompa giriÅŸinde (0=Error, 1=OK)
      PUMP_5_MANUAL_VALVE_STATUS : USInt := 1;   // Pump 5 Manual Valve - Tank-Pompa arasÄ± (0=KapalÄ±, 1=AÃ§Ä±k) ============================================================================= PUMP #6 VARIABLES (Pressure & Flow Control) =============================================================================
      PUMP_6_PRESSURE_SETPOINT : Real := 280.0;   // Pump 6 Pressure Setpoint (Bar) - Load Sensing coordinated
      PUMP_6_PRESSURE_ACTUAL : Real := 0.0;   // Pump 6 Actual Pressure (Bar) - Sensor feedback
      PUMP_6_FLOW_SETPOINT : Real := 30.0;   // Pump 6 Flow Setpoint (L/min) - User adjustable
      PUMP_6_FLOW_ACTUAL : Real := 0.0;   // Pump 6 Actual Flow (L/min) - Calculated value
      PUMP_6_LEAK_RATE : Real := 0.0;   // Pump 6 Leak Rate (L/min) - Diagnostic value
      PUMP_6_ENABLED : Bool := FALSE;   // Pump 6 Enable Control (PID enable) ============================================================================= MOTOR #6 VARIABLES (Electrical Parameters) =============================================================================
      MOTOR_6_RPM_SETPOINT : Real := 1000.0;   // Motor 6 Target RPM - VFD setpoint
      MOTOR_6_RPM_ACTUAL : Real := 0.0;   // Motor 6 Actual RPM - Encoder feedback
      MOTOR_6_CURRENT_A : Real := 0.0;   // Motor 6 Current (A) - Electrical measurement
      MOTOR_6_TEMPERATURE_C : Real := 25.0;   // Motor 6 Temperature (Â°C) - Thermal monitoring
      MOTOR_6_ENABLE : Bool := FALSE;   // Motor 6 Enable Control
      MOTOR_6_STATUS : USInt := 0;   // Motor 6 Status (0=Offline, 1=Ready, 2=Running, 3=Error)
      MOTOR_6_ERROR_CODE : USInt := 0;   // Motor 6 Error code - Diagnostic information
      MOTOR_6_START_CMD : Bool := FALSE;   // Motor 6 Start Command
      MOTOR_6_STOP_CMD : Bool := FALSE;   // Motor 6 Stop Command
      MOTOR_6_RESET_CMD : Bool := FALSE;   // Motor 6 Reset Command
      MOTOR_6_START_ACK : Bool := FALSE;   // Motor 6 Start Acknowledgment
      MOTOR_6_STOP_ACK : Bool := FALSE;   // Motor 6 Stop Acknowledgment
      MOTOR_6_RESET_ACK : Bool := FALSE;   // Motor 6 Reset Acknowledgment G120C FREE Telegram Variables - REMOVED (Use M8)
      MOTOR_6_CONTROL_WORD : Word;   // 200 : Word; // Motor 6 Control Word (PZD[0] Send)
      MOTOR_6_RPM_SETPOINT_WORD : Int;   // 202 : Int; // Motor 6 RPM Setpoint Word (PZD[1] Send)
      MOTOR_6_RESERVED_1 : Word;   // 204 : Word; // Motor 6 Reserved PZD[2] Send
      MOTOR_6_RESERVED_2 : Word;   // 206 : Word; // Motor 6 Reserved PZD[3] Send
      MOTOR_6_RESERVED_3 : Word;   // 208 : Word; // Motor 6 Reserved PZD[4] Send
      MOTOR_6_RESERVED_4 : Word;   // 210 : Word; // Motor 6 Reserved PZD[5] Send
      MOTOR_6_STATUS_WORD : Word;   // 200 : Word; // Motor 6 Status Word (PZD[0] Receive)
      MOTOR_6_RPM_ACTUAL_WORD : Int;   // 202 : Int; // Motor 6 RPM Actual Word (PZD[1] Receive)
      MOTOR_6_CURRENT_WORD : Int;   // 204 : Int; // Motor 6 Current Word (PZD[2] Receive)
      MOTOR_6_TEMPERATURE_WORD : Int;   // 206 : Int; // Motor 6 Temperature Word (PZD[3] Receive)
      MOTOR_6_ERROR_WORD : Word;   // 208 : Word; // Motor 6 Error/Warning Word (PZD[4] Receive)
      MOTOR_6_DIAGNOSTIC_WORD : Word;   // 210 : Word; // Motor 6 Diagnostic Word (PZD[5] Receive) ============================================================================= VALVE #6 VARIABLES (Position Control) =============================================================================
      VALVE_6_CURRENT_SETPOINT : Real := 0.0;   // Valve 6 Current Setpoint (0-10000) - Control output
      VALVE_6_CURRENT_MA : Real := 4.0;   // Valve 6 Current (4-20mA) - Analog signal
      PUMP_6_LINE_FILTER_STATUS : USInt := 2;   // Pump 6 Line Filter - Pompa Ã§Ä±kÄ±ÅŸÄ±nda (0=Error, 1=Warning, 2=OK)
      PUMP_6_SUCTION_FILTER_STATUS : USInt := 1;   // Pump 6 Suction Filter - Pompa giriÅŸinde (0=Error, 1=OK)
      PUMP_6_MANUAL_VALVE_STATUS : USInt := 1;   // Pump 6 Manual Valve - Tank-Pompa arasÄ± (0=KapalÄ±, 1=AÃ§Ä±k) ============================================================================= PUMP #7 VARIABLES (Fixed Displacement Motor - 1500 RPM, 34 L/min) =============================================================================
      PUMP_7_PRESSURE_SETPOINT : Real := 280.0;   // Pump 7 Pressure Setpoint (Bar) - Load Sensing coordinated
      PUMP_7_PRESSURE_ACTUAL : Real := 0.0;   // Pump 7 Actual Pressure (Bar) - Sensor feedback
      PUMP_7_FLOW_SETPOINT : Real := 34.0;   // Pump 7 Flow Setpoint (L/min) - Fixed displacement
      PUMP_7_FLOW_ACTUAL : Real := 0.0;   // Pump 7 Actual Flow (L/min) - Fixed at 34 L/min
      PUMP_7_LEAK_RATE : Real := 0.0;   // Pump 7 Leak Rate (L/min) - Diagnostic value
      PUMP_7_ENABLED : Bool := FALSE;   // Pump 7 Enable Control (PID enable) ============================================================================= MOTOR #7 VARIABLES (Fixed Displacement - 1500 RPM) =============================================================================
      MOTOR_7_RPM_SETPOINT : Real := 1500.0;   // Motor 7 Target RPM - Fixed displacement
      MOTOR_7_RPM_ACTUAL : Real := 0.0;   // Motor 7 Actual RPM - Fixed at 1500 RPM
      MOTOR_7_CURRENT_A : Real := 0.0;   // Motor 7 Current (A) - Electrical measurement
      MOTOR_7_TEMPERATURE_C : Real := 25.0;   // Motor 7 Temperature (Â°C) - Thermal monitoring
      MOTOR_7_ENABLE : Bool := FALSE;   // Motor 7 Enable Control
      MOTOR_7_STATUS : USInt := 0;   // Motor 7 Status (0=Offline, 1=Ready, 2=Running, 3=Error)
      MOTOR_7_ERROR_CODE : USInt := 0;   // Motor 7 Error code - Diagnostic information
      MOTOR_7_START_CMD : Bool := FALSE;   // Motor 7 Start Command
      MOTOR_7_STOP_CMD : Bool := FALSE;   // Motor 7 Stop Command
      MOTOR_7_RESET_CMD : Bool := FALSE;   // Motor 7 Reset Command ============================================================================= VALVE #7 VARIABLES (Position Control) =============================================================================
      VALVE_7_CURRENT_SETPOINT : Real := 0.0;   // Valve 7 Current Setpoint (0-10000) - Control output
      VALVE_7_CURRENT_MA : Real := 4.0;   // Valve 7 Current (4-20mA) - Analog signal
      PUMP_7_LINE_FILTER_STATUS : USInt := 2;   // Pump 7 Line Filter - Pompa Ã§Ä±kÄ±ÅŸÄ±nda (0=Error, 1=Warning, 2=OK)
      PUMP_7_SUCTION_FILTER_STATUS : USInt := 1;   // Pump 7 Suction Filter - Pompa giriÅŸinde (0=Error, 1=OK)
      PUMP_7_MANUAL_VALVE_STATUS : USInt := 1;   // Pump 7 Manual Valve - Tank-Pompa arasÄ± (0=KapalÄ±, 1=AÃ§Ä±k) ============================================================================= VALVE EXECUTION VARIABLES (Digital Control - Based on Git Analysis) =============================================================================
      VALVE_1_EXECUTION : USInt := 0;   // Valve 1 Digital Control (0=Closed, 1=Open)
      VALVE_2_EXECUTION : USInt := 0;   // Valve 2 Digital Control (0=Closed, 1=Open)
      VALVE_3_EXECUTION : USInt := 0;   // Valve 3 Digital Control (0=Closed, 1=Open)
      VALVE_4_EXECUTION : USInt := 0;   // Valve 4 Digital Control (0=Closed, 1=Open)
      VALVE_5_EXECUTION : USInt := 0;   // Valve 5 Digital Control (0=Closed, 1=Open)
      VALVE_6_EXECUTION : USInt := 0;   // Valve 6 Digital Control (0=Closed, 1=Open)
      VALVE_7_EXECUTION : USInt := 0;   // Valve 7 Digital Control (0=Closed, 1=Open) ============================================================================= LINE FILTER EXECUTION VARIABLES (Filter Status Control) =============================================================================
      LINE_FILTER_1_EXECUTION : USInt := 2;   // Motor 1 Line Filter (0=Error, 1=Warning, 2=OK)
      LINE_FILTER_2_EXECUTION : USInt := 2;   // Motor 2 Line Filter (0=Error, 1=Warning, 2=OK)
      LINE_FILTER_3_EXECUTION : USInt := 2;   // Motor 3 Line Filter (0=Error, 1=Warning, 2=OK)
      LINE_FILTER_4_EXECUTION : USInt := 2;   // Motor 4 Line Filter (0=Error, 1=Warning, 2=OK)
      LINE_FILTER_5_EXECUTION : USInt := 2;   // Motor 5 Line Filter (0=Error, 1=Warning, 2=OK)
      LINE_FILTER_6_EXECUTION : USInt := 2;   // Motor 6 Line Filter (0=Error, 1=Warning, 2=OK)
      LINE_FILTER_7_EXECUTION : USInt := 2;   // Motor 7 Line Filter (0=Error, 1=Warning, 2=OK) ============================================================================= SUCTION FILTER EXECUTION VARIABLES (Filter Status Control) =============================================================================
      SUCTION_FILTER_1_EXECUTION : USInt := 1;   // Motor 1 Suction Filter (0=Error, 1=OK)
      SUCTION_FILTER_2_EXECUTION : USInt := 1;   // Motor 2 Suction Filter (0=Error, 1=OK)
      SUCTION_FILTER_3_EXECUTION : USInt := 1;   // Motor 3 Suction Filter (0=Error, 1=OK)
      SUCTION_FILTER_4_EXECUTION : USInt := 1;   // Motor 4 Suction Filter (0=Error, 1=OK)
      SUCTION_FILTER_5_EXECUTION : USInt := 1;   // Motor 5 Suction Filter (0=Error, 1=OK)
      SUCTION_FILTER_6_EXECUTION : USInt := 1;   // Motor 6 Suction Filter (0=Error, 1=OK)
      SUCTION_FILTER_7_EXECUTION : USInt := 1;   // Motor 7 Suction Filter (0=Error, 1=OK) ============================================================================= FLOW CONTROL VARIABLES (Debi Metre Feedback) =============================================================================
      PUMP_1_FLOW_METER_VALUE : Real := 0.0;   // Motor 1 Flow Meter Reading (L/min)
      PUMP_1_FLOW_ERROR : Real := 0.0;   // Motor 1 Flow Error (L/min)
      PUMP_1_CONTROL_MODE : USInt := 0;   // Motor 1 Control Mode (0=Flow, 1=Pressure)
      PUMP_1_DISPLACEMENT : Real := 100.0;   // Motor 1 Displacement (cc/rev)
      PUMP_2_FLOW_METER_VALUE : Real := 0.0;   // Motor 2 Flow Meter Reading (L/min)
      PUMP_2_FLOW_ERROR : Real := 0.0;   // Motor 2 Flow Error (L/min)
      PUMP_2_CONTROL_MODE : USInt := 0;   // Motor 2 Control Mode (0=Flow, 1=Pressure)
      PUMP_2_DISPLACEMENT : Real := 100.0;   // Motor 2 Displacement (cc/rev)
      PUMP_3_FLOW_METER_VALUE : Real := 0.0;   // Motor 3 Flow Meter Reading (L/min)
      PUMP_3_FLOW_ERROR : Real := 0.0;   // Motor 3 Flow Error (L/min)
      PUMP_3_CONTROL_MODE : USInt := 0;   // Motor 3 Control Mode (0=Flow, 1=Pressure)
      PUMP_3_DISPLACEMENT : Real := 100.0;   // Motor 3 Displacement (cc/rev)
      PUMP_4_FLOW_METER_VALUE : Real := 0.0;   // Motor 4 Flow Meter Reading (L/min)
      PUMP_4_FLOW_ERROR : Real := 0.0;   // Motor 4 Flow Error (L/min)
      PUMP_4_CONTROL_MODE : USInt := 0;   // Motor 4 Control Mode (0=Flow, 1=Pressure)
      PUMP_4_DISPLACEMENT : Real := 100.0;   // Motor 4 Displacement (cc/rev)
      PUMP_5_FLOW_METER_VALUE : Real := 0.0;   // Motor 5 Flow Meter Reading (L/min)
      PUMP_5_FLOW_ERROR : Real := 0.0;   // Motor 5 Flow Error (L/min)
      PUMP_5_CONTROL_MODE : USInt := 0;   // Motor 5 Control Mode (0=Flow, 1=Pressure)
      PUMP_5_DISPLACEMENT : Real := 100.0;   // Motor 5 Displacement (cc/rev)
      PUMP_6_FLOW_METER_VALUE : Real := 0.0;   // Motor 6 Flow Meter Reading (L/min)
      PUMP_6_FLOW_ERROR : Real := 0.0;   // Motor 6 Flow Error (L/min)
      PUMP_6_CONTROL_MODE : USInt := 0;   // Motor 6 Control Mode (0=Flow, 1=Pressure)
      PUMP_6_DISPLACEMENT : Real := 100.0;   // Motor 6 Displacement (cc/rev)
      PUMP_7_FLOW_METER_VALUE : Real := 0.0;   // Motor 7 Flow Meter Reading (L/min)
      PUMP_7_CONTROL_MODE : USInt := 0;   // Motor 7 Control Mode (0=Flow, 1=Pressure)
      PUMP_7_DISPLACEMENT : Real := 34.0;   // Motor 7 Fixed Flow (L/min @ 1500 RPM) ============================================================================= MOTOR WEAR LEVELING VARIABLES (Motors 1-6 Only) =============================================================================
      WEAR_LEVELING_ENABLE : Bool := TRUE;   // Wear leveling algorithm enable/disable
      DEFAULT_MAINTENANCE_HOURS : Real := 1000.0;   // Default maintenance period (hours)
      MOTOR_1_OPERATING_HOURS : Real := 0.0;   // Motor 1 Total operating hours
      MOTOR_1_MAINTENANCE_HOURS : Real := 1000.0;   // Motor 1 Maintenance period
      MOTOR_1_MAINTENANCE_DUE : Bool := FALSE;   // Motor 1 Maintenance due flag
      MOTOR_1_LAST_MAINTENANCE_DATE : DTL;   // Motor 1 Last maintenance date
      MOTOR_1_SELECTION_PRIORITY : USInt := 0;   // Motor 1 Selection priority (0=highest)
      MOTOR_2_OPERATING_HOURS : Real := 0.0;   // Motor 2 Total operating hours
      MOTOR_2_MAINTENANCE_HOURS : Real := 1000.0;   // Motor 2 Maintenance period
      MOTOR_2_MAINTENANCE_DUE : Bool := FALSE;   // Motor 2 Maintenance due flag
      MOTOR_2_LAST_MAINTENANCE_DATE : DTL;   // Motor 2 Last maintenance date
      MOTOR_2_SELECTION_PRIORITY : USInt := 0;   // Motor 2 Selection priority (0=highest)
      MOTOR_3_OPERATING_HOURS : Real := 0.0;   // Motor 3 Total operating hours
      MOTOR_3_MAINTENANCE_HOURS : Real := 1000.0;   // Motor 3 Maintenance period
      MOTOR_3_MAINTENANCE_DUE : Bool := FALSE;   // Motor 3 Maintenance due flag
      MOTOR_3_LAST_MAINTENANCE_DATE : DTL;   // Motor 3 Last maintenance date
      MOTOR_3_SELECTION_PRIORITY : USInt := 0;   // Motor 3 Selection priority (0=highest)
      MOTOR_4_OPERATING_HOURS : Real := 0.0;   // Motor 4 Total operating hours
      MOTOR_4_MAINTENANCE_HOURS : Real := 1000.0;   // Motor 4 Maintenance period
      MOTOR_4_MAINTENANCE_DUE : Bool := FALSE;   // Motor 4 Maintenance due flag
      MOTOR_4_LAST_MAINTENANCE_DATE : DTL;   // Motor 4 Last maintenance date
      MOTOR_4_SELECTION_PRIORITY : USInt := 0;   // Motor 4 Selection priority (0=highest)
      MOTOR_5_OPERATING_HOURS : Real := 0.0;   // Motor 5 Total operating hours
      MOTOR_5_MAINTENANCE_HOURS : Real := 1000.0;   // Motor 5 Maintenance period
      MOTOR_5_MAINTENANCE_DUE : Bool := FALSE;   // Motor 5 Maintenance due flag
      MOTOR_5_LAST_MAINTENANCE_DATE : DTL;   // Motor 5 Last maintenance date
      MOTOR_5_SELECTION_PRIORITY : USInt := 0;   // Motor 5 Selection priority (0=highest)
      MOTOR_6_OPERATING_HOURS : Real := 0.0;   // Motor 6 Total operating hours
      MOTOR_6_MAINTENANCE_HOURS : Real := 1000.0;   // Motor 6 Maintenance period
      MOTOR_6_MAINTENANCE_DUE : Bool := FALSE;   // Motor 6 Maintenance due flag
      MOTOR_6_LAST_MAINTENANCE_DATE : DTL;   // Motor 6 Last maintenance date
      MOTOR_6_SELECTION_PRIORITY : USInt := 0;   // Motor 6 Selection priority (0=highest) Motor 7 Separate Tracking (Fixed Displacement)
      MOTOR_7_OPERATING_HOURS : Real := 0.0;   // Motor 7 Total operating hours
      MOTOR_7_MAINTENANCE_HOURS : Real := 1500.0;   // Motor 7 Maintenance period (longer for fixed)
      MOTOR_7_MAINTENANCE_DUE : Bool := FALSE;   // Motor 7 Maintenance due flag
      MOTOR_7_LAST_MAINTENANCE_DATE : DTL;   // Motor 7 Last maintenance date ============================================================================= VALVE RESPONSE TIME SETTINGS (Configurable) =============================================================================
      VALVE_RESPONSE_TIME : Time := T#40MS;   // Global valve response time (configurable)
      VALVE_RESPONSE_AUTO : Bool := FALSE;   // Automatic response time adjustment
      VALVE_RESPONSE_MIN : Time := T#20MS;   // Minimum response time limit
      VALVE_RESPONSE_MAX : Time := T#500MS;   // Maximum response time limit ============================================================================= AT ADDRESSING TEST VARIABLES - REMOVE AFTER TESTING =============================================================================
      AT_TEST_OUTPUT : Word;   // 90 : Word := 16#1234; // Test output word
      AT_TEST_INPUT : Word;   // 90 : Word; // Test input word
      AT_TEST_NORMAL : Word := 16#ABCD;   // Normal variable for comparison ============================================================================= CAN COMMUNICATION STATUS =============================================================================
      CAN_COMMUNICATION_ACTIVE : Bool := FALSE;   // CAN communication status
      CAN_TCP_CONNECTED : Bool := FALSE;   // TCP connection status
      CAN_TCP_IP_ADDRESS : String[15] := '192.168.100.21';   // Gateway IP
      CAN_TCP_PORT : UInt := 502;   // Gateway port
      CAN_ACTIVE_DEVICE_COUNT : USInt := 0;   // Number of responding devices
      CAN_SYSTEM_ERROR : Bool := FALSE;   // CAN communication error
   END_VAR
BEGIN
END_DATA_BLOCK

DATA_BLOCK "DB_System_Coordinator_Instance"   // DB2
TITLE = 'System Coordinator Instance DB - TIA Portal V17 Compatible'
{ S7_Optimized_Access := 'TRUE' }
AUTHOR : TUSAÅž HGU Control System
VERSION : 2.0
// =============================================================================
//  SYSTEM COORDINATOR INSTANCE DATA BLOCK - UPDATED
//  TIA Portal V17 Compatible Instance DB for System Level Coordination
//  Description: Load Sensing, Emergency Stop, System Status Management
//  =============================================================================
// stored: InstanceOfName FB_System_Coordinator
"FB_System_Coordinator"
BEGIN
END_DATA_BLOCK

FUNCTION_BLOCK "FB_System_Coordinator"   // FB1, SCL
{ S7_Optimized_Access := 'TRUE' }
VERSION : 2.0
// =============================================================================
//  TUSAÅž HGU System Coordinator V17 - UPDATED
//  Purpose: System-wide coordination with new algorithm integration
//  Features: Motor selection, dual control coordination, wear leveling
//  Motor 1-6: Variable displacement, Motor 7: Fixed displacement
//  =============================================================================
   VAR_INPUT
      Enable : Bool := FALSE;   // System enable from OB1
      SystemCommand : DInt := 0;   // System command from HMI System flow requirements
      System_Total_Flow_Setpoint : Real := 100.0;   // Total required flow (L/min)
   END_VAR
   VAR_OUTPUT
      SystemReady : Bool := FALSE;   // System ready status
      SystemError : Bool := FALSE;   // System error status
      SystemStatus : DInt := 0;   // System status code Coordination status
      Active_Motor_Count : USInt := 0;   // Number of active motors
      Total_System_Flow : Real := 0.0;   // Total system flow capacity
      System_Control_Mode : USInt := 0;   // Overall system control mode VAR_IN_OUT DB_HGU_Data : "DB_HGU_Execution_V17"; // Reference to main DB - Moved to direct access END_VAR Motor selection instance
   END_VAR
   VAR
      Motor_Selector : "FB_Motor_Selection";   // Motor selection algorithm Dual controller instances for each motor
      Dual_Controller_1 : "FB_Dual_Controller";
      Dual_Controller_2 : "FB_Dual_Controller";
      Dual_Controller_3 : "FB_Dual_Controller";
      Dual_Controller_4 : "FB_Dual_Controller";
      Dual_Controller_5 : "FB_Dual_Controller";
      Dual_Controller_6 : "FB_Dual_Controller";
      Dual_Controller_7 : "FB_Dual_Controller";   // Motor 7 fixed displacement G120C drive controller instances for Motors 1-6
      G120C_Drive_1 : "FB_G120C_Drive";   // Motor 1 G120C drive controller
      G120C_Drive_2 : "FB_G120C_Drive";   // Motor 2 G120C drive controller
      G120C_Drive_3 : "FB_G120C_Drive";   // Motor 3 G120C drive controller
      G120C_Drive_4 : "FB_G120C_Drive";   // Motor 4 G120C drive controller
      G120C_Drive_5 : "FB_G120C_Drive";   // Motor 5 G120C drive controller
      G120C_Drive_6 : "FB_G120C_Drive";   // Motor 6 G120C drive controller System state management
      InitComplete : Bool := FALSE;
      SystemTimer : TON_TIME;
      LastSystemSetpoint : Real := 0.0;
      SystemSetpointChanged : Bool := FALSE;   // Coordination variables
      i : USInt;
      ActivePumpCount : USInt := 0;
      TotalPressure : Real := 0.0;
      AveragePressure : Real := 0.0;
      Total_Flow_Capacity : Real := 0.0;   // System state machine
      SystemState : USInt := 0;   // 0=Init, 1=Ready, 2=Running, 3=Error
      StateTimer : TON_TIME;   // Motor hours tracking
      Hour_Update_Timer : TON_TIME;   // 1-minute timer for operating hours (more accurate)
      Motor_Running_Array : Array[1..7] of Bool;   // Motor running status Flow distribution for selected motors
      Flow_Per_Motor : Real := 0.0;   // Individual motor flow assignment
      Selected_Motor_Flow : Real := 0.0;   // Flow for variable motors only Error tracking
      System_Error_Code : USInt := 0;   // Detailed error code
      Controller_Errors : USInt := 0;   // Count of controller errors Pressure setpoint management
      Last_System_Pressure_Setpoint : Real := 0.0;   // Previous system pressure setpoint
      System_Pressure_Changed : Bool := FALSE;   // System pressure setpoint changed flag
   END_VAR
   VAR_TEMP
      Motor_Flow_Setpoint : Real;   // Temporary flow calculation
      Motor_Available : Bool;   // Temporary motor availability
   END_VAR
   // StateTimer.PT := T#2S;
   // Hour_Update_Timer.PT := T#1M;
BEGIN


   // =============================================================================
   // SYSTEM INITIALIZATION
   // =============================================================================
   IF NOT #InitComplete THEN
       "DB_HGU_Execution_V17".SYSTEM_STATUS := 0;          // System initializing
       "DB_HGU_Execution_V17".SYSTEM_PRESSURE_SETPOINT := 280.0; // Default setpoint

       // Initialize motor hours tracking
       #Hour_Update_Timer(IN := FALSE,
                          PT := T#60s);

       // Initialize motor running status
       FOR #i := 1 TO 7 DO
           #Motor_Running_Array[#i] := FALSE;
       END_FOR;

       #InitComplete := TRUE;
       #SystemState := 0;
   END_IF;

   // =============================================================================
   // MAIN SYSTEM LOGIC
   // =============================================================================
   IF #Enable THEN

       // =============================================================================
       // MOTOR SELECTION ALGORITHM WITH SAFETY INTEGRATION
       // =============================================================================
       #Motor_Selector(
                       Enable := TRUE,
                       Wear_Leveling_Enable := "DB_HGU_Execution_V17".WEAR_LEVELING_ENABLE,
                       Required_Total_Flow := #System_Total_Flow_Setpoint,

                       // Motor enable status
                       Motor_1_Enable := "DB_HGU_Execution_V17".MOTOR_1_ENABLE,
                       Motor_2_Enable := "DB_HGU_Execution_V17".MOTOR_2_ENABLE,
                       Motor_3_Enable := "DB_HGU_Execution_V17".MOTOR_3_ENABLE,
                       Motor_4_Enable := "DB_HGU_Execution_V17".MOTOR_4_ENABLE,
                       Motor_5_Enable := "DB_HGU_Execution_V17".MOTOR_5_ENABLE,
                       Motor_6_Enable := "DB_HGU_Execution_V17".MOTOR_6_ENABLE,
                       Motor_7_Enable := "DB_HGU_Execution_V17".MOTOR_7_ENABLE,

                       // Operating hours
                       Motor_1_Hours := "DB_HGU_Execution_V17".MOTOR_1_OPERATING_HOURS,
                       Motor_2_Hours := "DB_HGU_Execution_V17".MOTOR_2_OPERATING_HOURS,
                       Motor_3_Hours := "DB_HGU_Execution_V17".MOTOR_3_OPERATING_HOURS,
                       Motor_4_Hours := "DB_HGU_Execution_V17".MOTOR_4_OPERATING_HOURS,
                       Motor_5_Hours := "DB_HGU_Execution_V17".MOTOR_5_OPERATING_HOURS,
                       Motor_6_Hours := "DB_HGU_Execution_V17".MOTOR_6_OPERATING_HOURS,

                       // Maintenance status
                       Motor_1_Maintenance_Due := "DB_HGU_Execution_V17".MOTOR_1_MAINTENANCE_DUE,
                       Motor_2_Maintenance_Due := "DB_HGU_Execution_V17".MOTOR_2_MAINTENANCE_DUE,
                       Motor_3_Maintenance_Due := "DB_HGU_Execution_V17".MOTOR_3_MAINTENANCE_DUE,
                       Motor_4_Maintenance_Due := "DB_HGU_Execution_V17".MOTOR_4_MAINTENANCE_DUE,
                       Motor_5_Maintenance_Due := "DB_HGU_Execution_V17".MOTOR_5_MAINTENANCE_DUE,
                       Motor_6_Maintenance_Due := "DB_HGU_Execution_V17".MOTOR_6_MAINTENANCE_DUE,

                       // Safety status inputs (Pump 1-7)
                       Pump_1_Line_Filter_Status := "DB_HGU_Execution_V17".PUMP_1_LINE_FILTER_STATUS,
                       Pump_1_Suction_Filter_Status := "DB_HGU_Execution_V17".PUMP_1_SUCTION_FILTER_STATUS,
                       Pump_1_Manual_Valve_Status := "DB_HGU_Execution_V17".PUMP_1_MANUAL_VALVE_STATUS,

                       Pump_2_Line_Filter_Status := "DB_HGU_Execution_V17".PUMP_2_LINE_FILTER_STATUS,
                       Pump_2_Suction_Filter_Status := "DB_HGU_Execution_V17".PUMP_2_SUCTION_FILTER_STATUS,
                       Pump_2_Manual_Valve_Status := "DB_HGU_Execution_V17".PUMP_2_MANUAL_VALVE_STATUS,

                       Pump_3_Line_Filter_Status := "DB_HGU_Execution_V17".PUMP_3_LINE_FILTER_STATUS,
                       Pump_3_Suction_Filter_Status := "DB_HGU_Execution_V17".PUMP_3_SUCTION_FILTER_STATUS,
                       Pump_3_Manual_Valve_Status := "DB_HGU_Execution_V17".PUMP_3_MANUAL_VALVE_STATUS,

                       Pump_4_Line_Filter_Status := "DB_HGU_Execution_V17".PUMP_4_LINE_FILTER_STATUS,
                       Pump_4_Suction_Filter_Status := "DB_HGU_Execution_V17".PUMP_4_SUCTION_FILTER_STATUS,
                       Pump_4_Manual_Valve_Status := "DB_HGU_Execution_V17".PUMP_4_MANUAL_VALVE_STATUS,

                       Pump_5_Line_Filter_Status := "DB_HGU_Execution_V17".PUMP_5_LINE_FILTER_STATUS,
                       Pump_5_Suction_Filter_Status := "DB_HGU_Execution_V17".PUMP_5_SUCTION_FILTER_STATUS,
                       Pump_5_Manual_Valve_Status := "DB_HGU_Execution_V17".PUMP_5_MANUAL_VALVE_STATUS,

                       Pump_6_Line_Filter_Status := "DB_HGU_Execution_V17".PUMP_6_LINE_FILTER_STATUS,
                       Pump_6_Suction_Filter_Status := "DB_HGU_Execution_V17".PUMP_6_SUCTION_FILTER_STATUS,
                       Pump_6_Manual_Valve_Status := "DB_HGU_Execution_V17".PUMP_6_MANUAL_VALVE_STATUS,

                       Pump_7_Line_Filter_Status := "DB_HGU_Execution_V17".PUMP_7_LINE_FILTER_STATUS,
                       Pump_7_Suction_Filter_Status := "DB_HGU_Execution_V17".PUMP_7_SUCTION_FILTER_STATUS,
                       Pump_7_Manual_Valve_Status := "DB_HGU_Execution_V17".PUMP_7_MANUAL_VALVE_STATUS,

                       // System parameters
                       Motor_Displacement := 100.0,           // cc/rev
                       Max_Motor_RPM := 1500.0,              // RPM
                       Motor_7_Fixed_Flow := 34.0            // L/min
       );

       // =============================================================================
       // FLOW DISTRIBUTION CALCULATION
       // =============================================================================

       // Calculate flow for variable motors (excluding Motor 7)
       #Selected_Motor_Flow := #System_Total_Flow_Setpoint;
       IF #Motor_Selector.Motor_7_Selected THEN
           #Selected_Motor_Flow := #Selected_Motor_Flow - 34.0; // Subtract Motor 7 flow
       END_IF;

       // Ensure non-negative flow
       IF #Selected_Motor_Flow < 0.0 THEN
           #Selected_Motor_Flow := 0.0;
       END_IF;

       // Calculate flow per selected motor
       IF #Motor_Selector.Selected_Motor_Count > 0 THEN
           #Flow_Per_Motor := #Selected_Motor_Flow / USINT_TO_REAL(#Motor_Selector.Selected_Motor_Count);
       ELSE
           #Flow_Per_Motor := 0.0;
       END_IF;

       // =============================================================================
       // DUAL CONTROLLER COORDINATION (Motors 1-6)
       // =============================================================================

       // Motor 1 Dual Controller
       #Dual_Controller_1(
                          Enable := TRUE,
                          Motor_Enable := #Motor_Selector.Motor_1_Selected,
                          Pressure_Setpoint := "DB_HGU_Execution_V17".PUMP_1_PRESSURE_SETPOINT,
                          Pressure_Actual := "DB_HGU_Execution_V17".PUMP_1_PRESSURE_ACTUAL,
                          Flow_Setpoint := #Flow_Per_Motor,
                          Flow_Actual := "DB_HGU_Execution_V17".PUMP_1_FLOW_METER_VALUE,
                          Motor_Displacement := "DB_HGU_Execution_V17".PUMP_1_DISPLACEMENT,
                          Motor_Number := 1,
                          Valve_Response_Time := "DB_HGU_Execution_V17".VALVE_RESPONSE_TIME
       );

       // Update outputs for Motor 1
       "DB_HGU_Execution_V17".MOTOR_1_RPM_SETPOINT := #Dual_Controller_1.Motor_RPM;
       "DB_HGU_Execution_V17".VALVE_1_CURRENT_SETPOINT := #Dual_Controller_1.Valve_Current;
       // "DB_HGU_Execution_V17".PUMP_1_CONTROL_MODE := 0; // Manual mode assignment if needed
       #Motor_Running_Array[1] := #G120C_Drive_1.Motor_Running;

       // Motor 2 Dual Controller
       #Dual_Controller_2(
                          Enable := TRUE,
                          Motor_Enable := #Motor_Selector.Motor_2_Selected,
                          Pressure_Setpoint := "DB_HGU_Execution_V17".PUMP_2_PRESSURE_SETPOINT,
                          Pressure_Actual := "DB_HGU_Execution_V17".PUMP_2_PRESSURE_ACTUAL,
                          Flow_Setpoint := #Flow_Per_Motor,
                          Flow_Actual := "DB_HGU_Execution_V17".PUMP_2_FLOW_METER_VALUE,
                          Motor_Displacement := "DB_HGU_Execution_V17".PUMP_2_DISPLACEMENT,
                          Motor_Number := 2,
                          Valve_Response_Time := "DB_HGU_Execution_V17".VALVE_RESPONSE_TIME
       );

       "DB_HGU_Execution_V17".MOTOR_2_RPM_SETPOINT := #Dual_Controller_2.Motor_RPM;
       "DB_HGU_Execution_V17".VALVE_2_CURRENT_SETPOINT := #Dual_Controller_2.Valve_Current;
       // "DB_HGU_Execution_V17".PUMP_2_CONTROL_MODE := 0; // Manual mode assignment if needed
       #Motor_Running_Array[2] := #G120C_Drive_2.Motor_Running;

       // Motor 3 Dual Controller
       #Dual_Controller_3(
                          Enable := TRUE,
                          Motor_Enable := #Motor_Selector.Motor_3_Selected,
                          Pressure_Setpoint := "DB_HGU_Execution_V17".PUMP_3_PRESSURE_SETPOINT,
                          Pressure_Actual := "DB_HGU_Execution_V17".PUMP_3_PRESSURE_ACTUAL,
                          Flow_Setpoint := #Flow_Per_Motor,
                          Flow_Actual := "DB_HGU_Execution_V17".PUMP_3_FLOW_METER_VALUE,
                          Motor_Displacement := "DB_HGU_Execution_V17".PUMP_3_DISPLACEMENT,
                          Motor_Number := 3,
                          Valve_Response_Time := "DB_HGU_Execution_V17".VALVE_RESPONSE_TIME
       );

       "DB_HGU_Execution_V17".MOTOR_3_RPM_SETPOINT := #Dual_Controller_3.Motor_RPM;
       "DB_HGU_Execution_V17".VALVE_3_CURRENT_SETPOINT := #Dual_Controller_3.Valve_Current;
       // "DB_HGU_Execution_V17".PUMP_3_CONTROL_MODE := 0; // Manual mode assignment if needed
       #Motor_Running_Array[3] := #G120C_Drive_3.Motor_Running;

       // Motor 4 Dual Controller
       #Dual_Controller_4(
                          Enable := TRUE,
                          Motor_Enable := #Motor_Selector.Motor_4_Selected,
                          Pressure_Setpoint := "DB_HGU_Execution_V17".PUMP_4_PRESSURE_SETPOINT,
                          Pressure_Actual := "DB_HGU_Execution_V17".PUMP_4_PRESSURE_ACTUAL,
                          Flow_Setpoint := #Flow_Per_Motor,
                          Flow_Actual := "DB_HGU_Execution_V17".PUMP_4_FLOW_METER_VALUE,
                          Motor_Displacement := "DB_HGU_Execution_V17".PUMP_4_DISPLACEMENT,
                          Motor_Number := 4,
                          Valve_Response_Time := "DB_HGU_Execution_V17".VALVE_RESPONSE_TIME
       );

       "DB_HGU_Execution_V17".MOTOR_4_RPM_SETPOINT := #Dual_Controller_4.Motor_RPM;
       "DB_HGU_Execution_V17".VALVE_4_CURRENT_SETPOINT := #Dual_Controller_4.Valve_Current;
       // "DB_HGU_Execution_V17".PUMP_4_CONTROL_MODE := 0; // Manual mode assignment if needed
       #Motor_Running_Array[4] := #G120C_Drive_4.Motor_Running;

       // Motor 5 Dual Controller
       #Dual_Controller_5(
                          Enable := TRUE,
                          Motor_Enable := #Motor_Selector.Motor_5_Selected,
                          Pressure_Setpoint := "DB_HGU_Execution_V17".PUMP_5_PRESSURE_SETPOINT,
                          Pressure_Actual := "DB_HGU_Execution_V17".PUMP_5_PRESSURE_ACTUAL,
                          Flow_Setpoint := #Flow_Per_Motor,
                          Flow_Actual := "DB_HGU_Execution_V17".PUMP_5_FLOW_METER_VALUE,
                          Motor_Displacement := "DB_HGU_Execution_V17".PUMP_5_DISPLACEMENT,
                          Motor_Number := 5,
                          Valve_Response_Time := "DB_HGU_Execution_V17".VALVE_RESPONSE_TIME
       );

       "DB_HGU_Execution_V17".MOTOR_5_RPM_SETPOINT := #Dual_Controller_5.Motor_RPM;
       "DB_HGU_Execution_V17".VALVE_5_CURRENT_SETPOINT := #Dual_Controller_5.Valve_Current;
       // "DB_HGU_Execution_V17".PUMP_5_CONTROL_MODE := 0; // Manual mode assignment if needed
       #Motor_Running_Array[5] := #G120C_Drive_5.Motor_Running;

       // Motor 6 Dual Controller
       #Dual_Controller_6(
                          Enable := TRUE,
                          Motor_Enable := #Motor_Selector.Motor_6_Selected,
                          Pressure_Setpoint := "DB_HGU_Execution_V17".PUMP_6_PRESSURE_SETPOINT,
                          Pressure_Actual := "DB_HGU_Execution_V17".PUMP_6_PRESSURE_ACTUAL,
                          Flow_Setpoint := #Flow_Per_Motor,
                          Flow_Actual := "DB_HGU_Execution_V17".PUMP_6_FLOW_METER_VALUE,
                          Motor_Displacement := "DB_HGU_Execution_V17".PUMP_6_DISPLACEMENT,
                          Motor_Number := 6,
                          Valve_Response_Time := "DB_HGU_Execution_V17".VALVE_RESPONSE_TIME
       );

       "DB_HGU_Execution_V17".MOTOR_6_RPM_SETPOINT := #Dual_Controller_6.Motor_RPM;
       "DB_HGU_Execution_V17".VALVE_6_CURRENT_SETPOINT := #Dual_Controller_6.Valve_Current;
       // "DB_HGU_Execution_V17".PUMP_6_CONTROL_MODE := 0; // Manual mode assignment if needed
       #Motor_Running_Array[6] := #G120C_Drive_6.Motor_Running;

       // =============================================================================
       // G120C DRIVE CONTROL (Motors 1-6)
       // =============================================================================

       // Motor 1 G120C Drive Controller
       #G120C_Drive_1(
                      Enable := #Motor_Selector.Motor_1_Selected,
                      Motor_Number := 1,
                      RPM_Setpoint := #Dual_Controller_1.Motor_RPM,
                      Start_Command := "DB_HGU_Execution_V17".MOTOR_1_START_CMD,
                      Stop_Command := "DB_HGU_Execution_V17".MOTOR_1_STOP_CMD,
                      Reset_Command := "DB_HGU_Execution_V17".MOTOR_1_RESET_CMD,
                      Emergency_Stop := "DB_HGU_Execution_V17".EMERGENCY_STOP,
                      Motor_Enable_Switch := "DB_HGU_Execution_V17".MOTOR_1_ENABLE,
                      Max_RPM := 1500.0,
                      Ramp_Up_Time := T#5s,
                      Ramp_Down_Time := T#3s,
                      Control_Word := "M1_Control_Word",
                      Status_Word := "M1_Status_Word",
                      RPM_Setpoint_Word := "M1_RPM_Setpoint_Word",
                      RPM_Actual_Word := "M1_RPM_Actual_Word",
                      Current_Word := "M1_Current_Word",
                      Temperature_Word := "M1_Temperature_Word",
                      Error_Word := "M1_Error_Word"
       );

       // Update Motor 1 outputs from G120C
       "DB_HGU_Execution_V17".MOTOR_1_STATUS := BOOL_TO_USINT(#G120C_Drive_1.Motor_Running) * 2;
       "DB_HGU_Execution_V17".MOTOR_1_RPM_ACTUAL := #G120C_Drive_1.RPM_Actual;
       "DB_HGU_Execution_V17".MOTOR_1_CURRENT_A := #G120C_Drive_1.Current_A;
       "DB_HGU_Execution_V17".MOTOR_1_TEMPERATURE_C := #G120C_Drive_1.Temperature_C;
       "DB_HGU_Execution_V17".MOTOR_1_ERROR_CODE := #G120C_Drive_1.Error_Code;
       "DB_HGU_Execution_V17".MOTOR_1_START_ACK := #G120C_Drive_1.Start_Ack;
       "DB_HGU_Execution_V17".MOTOR_1_STOP_ACK := #G120C_Drive_1.Stop_Ack;
       "DB_HGU_Execution_V17".MOTOR_1_RESET_ACK := #G120C_Drive_1.Reset_Ack;

       // Motor 2 G120C Drive Controller
       #G120C_Drive_2(
                      Enable := #Motor_Selector.Motor_2_Selected,
                      Motor_Number := 2,
                      RPM_Setpoint := #Dual_Controller_2.Motor_RPM,
                      Start_Command := "DB_HGU_Execution_V17".MOTOR_2_START_CMD,
                      Stop_Command := "DB_HGU_Execution_V17".MOTOR_2_STOP_CMD,
                      Reset_Command := "DB_HGU_Execution_V17".MOTOR_2_RESET_CMD,
                      Emergency_Stop := "DB_HGU_Execution_V17".EMERGENCY_STOP,
                      Motor_Enable_Switch := "DB_HGU_Execution_V17".MOTOR_2_ENABLE,
                      Max_RPM := 1500.0,
                      Ramp_Up_Time := T#5s,
                      Ramp_Down_Time := T#3s,
                      Control_Word := "M2_Control_Word",
                      Status_Word := "M2_Status_Word",
                      RPM_Setpoint_Word := "M2_RPM_Setpoint_Word",
                      RPM_Actual_Word := "M2_RPM_Actual_Word",
                      Current_Word := "M2_Current_Word",
                      Temperature_Word := "M2_Temperature_Word",
                      Error_Word := "M2_Error_Word"
       );

       "DB_HGU_Execution_V17".MOTOR_2_STATUS := BOOL_TO_USINT(#G120C_Drive_2.Motor_Running) * 2;
       "DB_HGU_Execution_V17".MOTOR_2_RPM_ACTUAL := #G120C_Drive_2.RPM_Actual;
       "DB_HGU_Execution_V17".MOTOR_2_CURRENT_A := #G120C_Drive_2.Current_A;
       "DB_HGU_Execution_V17".MOTOR_2_TEMPERATURE_C := #G120C_Drive_2.Temperature_C;
       "DB_HGU_Execution_V17".MOTOR_2_ERROR_CODE := #G120C_Drive_2.Error_Code;
       "DB_HGU_Execution_V17".MOTOR_2_START_ACK := #G120C_Drive_2.Start_Ack;
       "DB_HGU_Execution_V17".MOTOR_2_STOP_ACK := #G120C_Drive_2.Stop_Ack;
       "DB_HGU_Execution_V17".MOTOR_2_RESET_ACK := #G120C_Drive_2.Reset_Ack;

       // Motor 3 G120C Drive Controller
       #G120C_Drive_3(
                      Enable := #Motor_Selector.Motor_3_Selected,
                      Motor_Number := 3,
                      RPM_Setpoint := #Dual_Controller_3.Motor_RPM,
                      Start_Command := "DB_HGU_Execution_V17".MOTOR_3_START_CMD,
                      Stop_Command := "DB_HGU_Execution_V17".MOTOR_3_STOP_CMD,
                      Reset_Command := "DB_HGU_Execution_V17".MOTOR_3_RESET_CMD,
                      Emergency_Stop := "DB_HGU_Execution_V17".EMERGENCY_STOP,
                      Motor_Enable_Switch := "DB_HGU_Execution_V17".MOTOR_3_ENABLE,
                      Max_RPM := 1500.0,
                      Ramp_Up_Time := T#5s,
                      Ramp_Down_Time := T#3s,
                      Control_Word := "M3_Control_Word",
                      Status_Word := "M3_Status_Word",
                      RPM_Setpoint_Word := "M3_RPM_Setpoint_Word",
                      RPM_Actual_Word := "M3_RPM_Actual_Word",
                      Current_Word := "M3_Current_Word",
                      Temperature_Word := "M3_Temperature_Word",
                      Error_Word := "M3_Error_Word"
       );

       "DB_HGU_Execution_V17".MOTOR_3_STATUS := BOOL_TO_USINT(#G120C_Drive_3.Motor_Running) * 2;
       "DB_HGU_Execution_V17".MOTOR_3_RPM_ACTUAL := #G120C_Drive_3.RPM_Actual;
       "DB_HGU_Execution_V17".MOTOR_3_CURRENT_A := #G120C_Drive_3.Current_A;
       "DB_HGU_Execution_V17".MOTOR_3_TEMPERATURE_C := #G120C_Drive_3.Temperature_C;
       "DB_HGU_Execution_V17".MOTOR_3_ERROR_CODE := #G120C_Drive_3.Error_Code;
       "DB_HGU_Execution_V17".MOTOR_3_START_ACK := #G120C_Drive_3.Start_Ack;
       "DB_HGU_Execution_V17".MOTOR_3_STOP_ACK := #G120C_Drive_3.Stop_Ack;
       "DB_HGU_Execution_V17".MOTOR_3_RESET_ACK := #G120C_Drive_3.Reset_Ack;

       // Motor 4 G120C Drive Controller
       #G120C_Drive_4(
                      Enable := #Motor_Selector.Motor_4_Selected,
                      Motor_Number := 4,
                      RPM_Setpoint := #Dual_Controller_4.Motor_RPM,
                      Start_Command := "DB_HGU_Execution_V17".MOTOR_4_START_CMD,
                      Stop_Command := "DB_HGU_Execution_V17".MOTOR_4_STOP_CMD,
                      Reset_Command := "DB_HGU_Execution_V17".MOTOR_4_RESET_CMD,
                      Emergency_Stop := "DB_HGU_Execution_V17".EMERGENCY_STOP,
                      Motor_Enable_Switch := "DB_HGU_Execution_V17".MOTOR_4_ENABLE,
                      Max_RPM := 1500.0,
                      Ramp_Up_Time := T#5s,
                      Ramp_Down_Time := T#3s,
                      Control_Word := "M4_Control_Word",
                      Status_Word := "M4_Status_Word",
                      RPM_Setpoint_Word := "M4_RPM_Setpoint_Word",
                      RPM_Actual_Word := "M4_RPM_Actual_Word",
                      Current_Word := "M4_Current_Word",
                      Temperature_Word := "M4_Temperature_Word",
                      Error_Word := "M4_Error_Word"
       );

       "DB_HGU_Execution_V17".MOTOR_4_STATUS := BOOL_TO_USINT(#G120C_Drive_4.Motor_Running) * 2;
       "DB_HGU_Execution_V17".MOTOR_4_RPM_ACTUAL := #G120C_Drive_4.RPM_Actual;
       "DB_HGU_Execution_V17".MOTOR_4_CURRENT_A := #G120C_Drive_4.Current_A;
       "DB_HGU_Execution_V17".MOTOR_4_TEMPERATURE_C := #G120C_Drive_4.Temperature_C;
       "DB_HGU_Execution_V17".MOTOR_4_ERROR_CODE := #G120C_Drive_4.Error_Code;
       "DB_HGU_Execution_V17".MOTOR_4_START_ACK := #G120C_Drive_4.Start_Ack;
       "DB_HGU_Execution_V17".MOTOR_4_STOP_ACK := #G120C_Drive_4.Stop_Ack;
       "DB_HGU_Execution_V17".MOTOR_4_RESET_ACK := #G120C_Drive_4.Reset_Ack;

       // Motor 5 G120C Drive Controller
       #G120C_Drive_5(
                      Enable := #Motor_Selector.Motor_5_Selected,
                      Motor_Number := 5,
                      RPM_Setpoint := #Dual_Controller_5.Motor_RPM,
                      Start_Command := "DB_HGU_Execution_V17".MOTOR_5_START_CMD,
                      Stop_Command := "DB_HGU_Execution_V17".MOTOR_5_STOP_CMD,
                      Reset_Command := "DB_HGU_Execution_V17".MOTOR_5_RESET_CMD,
                      Emergency_Stop := "DB_HGU_Execution_V17".EMERGENCY_STOP,
                      Motor_Enable_Switch := "DB_HGU_Execution_V17".MOTOR_5_ENABLE,
                      Max_RPM := 1500.0,
                      Ramp_Up_Time := T#5s,
                      Ramp_Down_Time := T#3s,
                      Control_Word := "M5_Control_Word",
                      Status_Word := "M5_Status_Word",
                      RPM_Setpoint_Word := "M5_RPM_Setpoint_Word",
                      RPM_Actual_Word := "M5_RPM_Actual_Word",
                      Current_Word := "M5_Current_Word",
                      Temperature_Word := "M5_Temperature_Word",
                      Error_Word := "M5_Error_Word"
       );

       "DB_HGU_Execution_V17".MOTOR_5_STATUS := BOOL_TO_USINT(#G120C_Drive_5.Motor_Running) * 2;
       "DB_HGU_Execution_V17".MOTOR_5_RPM_ACTUAL := #G120C_Drive_5.RPM_Actual;
       "DB_HGU_Execution_V17".MOTOR_5_CURRENT_A := #G120C_Drive_5.Current_A;
       "DB_HGU_Execution_V17".MOTOR_5_TEMPERATURE_C := #G120C_Drive_5.Temperature_C;
       "DB_HGU_Execution_V17".MOTOR_5_ERROR_CODE := #G120C_Drive_5.Error_Code;
       "DB_HGU_Execution_V17".MOTOR_5_START_ACK := #G120C_Drive_5.Start_Ack;
       "DB_HGU_Execution_V17".MOTOR_5_STOP_ACK := #G120C_Drive_5.Stop_Ack;
       "DB_HGU_Execution_V17".MOTOR_5_RESET_ACK := #G120C_Drive_5.Reset_Ack;

       // Motor 6 G120C Drive Controller
       #G120C_Drive_6(
                      Enable := #Motor_Selector.Motor_6_Selected,
                      Motor_Number := 6,
                      RPM_Setpoint := #Dual_Controller_6.Motor_RPM,
                      Start_Command := "DB_HGU_Execution_V17".MOTOR_6_START_CMD,
                      Stop_Command := "DB_HGU_Execution_V17".MOTOR_6_STOP_CMD,
                      Reset_Command := "DB_HGU_Execution_V17".MOTOR_6_RESET_CMD,
                      Emergency_Stop := "DB_HGU_Execution_V17".EMERGENCY_STOP,
                      Motor_Enable_Switch := "DB_HGU_Execution_V17".MOTOR_6_ENABLE,
                      Max_RPM := 1500.0,
                      Ramp_Up_Time := T#5s,
                      Ramp_Down_Time := T#3s,
                      Control_Word := "M6_Control_Word",
                      Status_Word := "M6_Status_Word",
                      RPM_Setpoint_Word := "M6_RPM_Setpoint_Word",
                      RPM_Actual_Word := "M6_RPM_Actual_Word",
                      Current_Word := "M6_Current_Word",
                      Temperature_Word := "M6_Temperature_Word",
                      Error_Word := "M6_Error_Word"
       );

       "DB_HGU_Execution_V17".MOTOR_6_STATUS := BOOL_TO_USINT(#G120C_Drive_6.Motor_Running) * 2;
       "DB_HGU_Execution_V17".MOTOR_6_RPM_ACTUAL := #G120C_Drive_6.RPM_Actual;
       "DB_HGU_Execution_V17".MOTOR_6_CURRENT_A := #G120C_Drive_6.Current_A;
       "DB_HGU_Execution_V17".MOTOR_6_TEMPERATURE_C := #G120C_Drive_6.Temperature_C;
       "DB_HGU_Execution_V17".MOTOR_6_ERROR_CODE := #G120C_Drive_6.Error_Code;
       "DB_HGU_Execution_V17".MOTOR_6_START_ACK := #G120C_Drive_6.Start_Ack;
       "DB_HGU_Execution_V17".MOTOR_6_STOP_ACK := #G120C_Drive_6.Stop_Ack;
       "DB_HGU_Execution_V17".MOTOR_6_RESET_ACK := #G120C_Drive_6.Reset_Ack;

       // =============================================================================
       // MOTOR 7 FIXED DISPLACEMENT CONTROL
       // =============================================================================
       #Dual_Controller_7(
                          Enable := TRUE,
                          Motor_Enable := #Motor_Selector.Motor_7_Selected,
                          Pressure_Setpoint := "DB_HGU_Execution_V17".PUMP_7_PRESSURE_SETPOINT,
                          Pressure_Actual := "DB_HGU_Execution_V17".PUMP_7_PRESSURE_ACTUAL,
                          Flow_Setpoint := 34.0,                // Fixed flow for Motor 7
                          Flow_Actual := "DB_HGU_Execution_V17".PUMP_7_FLOW_METER_VALUE,
                          Motor_Displacement := 34.0,           // Fixed displacement equivalent
                          Motor_Number := 7,
                          Valve_Response_Time := "DB_HGU_Execution_V17".VALVE_RESPONSE_TIME
       );

       // Motor 7 always runs at 1500 RPM when selected
       IF #Motor_Selector.Motor_7_Selected THEN
           "DB_HGU_Execution_V17".MOTOR_7_RPM_SETPOINT := 1500.0;
       ELSE
           "DB_HGU_Execution_V17".MOTOR_7_RPM_SETPOINT := 0.0;
       END_IF;

       "DB_HGU_Execution_V17".VALVE_7_CURRENT_SETPOINT := #Dual_Controller_7.Valve_Current;
       // "DB_HGU_Execution_V17".PUMP_7_CONTROL_MODE := 0; // Manual mode assignment if needed
       #Motor_Running_Array[7] := #Motor_Selector.Motor_7_Selected;

       // =============================================================================
       // MOTOR OPERATING HOURS TRACKING
       // =============================================================================
       #Hour_Update_Timer(IN := TRUE,
                          PT := T#60s); // 1 minute timer for accurate tracking

       IF #Hour_Update_Timer.Q THEN
           // Update operating hours for running motors (1 minute = 1/60 hour)
           IF #Motor_Running_Array[1] THEN
               "DB_HGU_Execution_V17".MOTOR_1_OPERATING_HOURS := "DB_HGU_Execution_V17".MOTOR_1_OPERATING_HOURS + 0.0167;
           END_IF;
           IF #Motor_Running_Array[2] THEN
               "DB_HGU_Execution_V17".MOTOR_2_OPERATING_HOURS := "DB_HGU_Execution_V17".MOTOR_2_OPERATING_HOURS + 0.0167;
           END_IF;
           IF #Motor_Running_Array[3] THEN
               "DB_HGU_Execution_V17".MOTOR_3_OPERATING_HOURS := "DB_HGU_Execution_V17".MOTOR_3_OPERATING_HOURS + 0.0167;
           END_IF;
           IF #Motor_Running_Array[4] THEN
               "DB_HGU_Execution_V17".MOTOR_4_OPERATING_HOURS := "DB_HGU_Execution_V17".MOTOR_4_OPERATING_HOURS + 0.0167;
           END_IF;
           IF #Motor_Running_Array[5] THEN
               "DB_HGU_Execution_V17".MOTOR_5_OPERATING_HOURS := "DB_HGU_Execution_V17".MOTOR_5_OPERATING_HOURS + 0.0167;
           END_IF;
           IF #Motor_Running_Array[6] THEN
               "DB_HGU_Execution_V17".MOTOR_6_OPERATING_HOURS := "DB_HGU_Execution_V17".MOTOR_6_OPERATING_HOURS + 0.0167;
           END_IF;
           IF #Motor_Running_Array[7] THEN
               "DB_HGU_Execution_V17".MOTOR_7_OPERATING_HOURS := "DB_HGU_Execution_V17".MOTOR_7_OPERATING_HOURS + 0.0167;
           END_IF;

           // Check maintenance due status
           "DB_HGU_Execution_V17".MOTOR_1_MAINTENANCE_DUE := ("DB_HGU_Execution_V17".MOTOR_1_OPERATING_HOURS >= "DB_HGU_Execution_V17".MOTOR_1_MAINTENANCE_HOURS);
           "DB_HGU_Execution_V17".MOTOR_2_MAINTENANCE_DUE := ("DB_HGU_Execution_V17".MOTOR_2_OPERATING_HOURS >= "DB_HGU_Execution_V17".MOTOR_2_MAINTENANCE_HOURS);
           "DB_HGU_Execution_V17".MOTOR_3_MAINTENANCE_DUE := ("DB_HGU_Execution_V17".MOTOR_3_OPERATING_HOURS >= "DB_HGU_Execution_V17".MOTOR_3_MAINTENANCE_HOURS);
           "DB_HGU_Execution_V17".MOTOR_4_MAINTENANCE_DUE := ("DB_HGU_Execution_V17".MOTOR_4_OPERATING_HOURS >= "DB_HGU_Execution_V17".MOTOR_4_MAINTENANCE_HOURS);
           "DB_HGU_Execution_V17".MOTOR_5_MAINTENANCE_DUE := ("DB_HGU_Execution_V17".MOTOR_5_OPERATING_HOURS >= "DB_HGU_Execution_V17".MOTOR_5_MAINTENANCE_HOURS);
           "DB_HGU_Execution_V17".MOTOR_6_MAINTENANCE_DUE := ("DB_HGU_Execution_V17".MOTOR_6_OPERATING_HOURS >= "DB_HGU_Execution_V17".MOTOR_6_MAINTENANCE_HOURS);
           "DB_HGU_Execution_V17".MOTOR_7_MAINTENANCE_DUE := ("DB_HGU_Execution_V17".MOTOR_7_OPERATING_HOURS >= "DB_HGU_Execution_V17".MOTOR_7_MAINTENANCE_HOURS);

           #Hour_Update_Timer(IN := FALSE,
                              PT := T#60s); // Reset timer
       END_IF;

       // =============================================================================
       // SAFETY MONITORING AND ERROR DETECTION
       // =============================================================================

       // Reset safety error counters
       #Controller_Errors := 0;
       #System_Error_Code := 0;

       // Check each motor's safety status and count safety violations
       FOR #i := 1 TO 7 DO
           CASE #i OF
               1:
                   IF ("DB_HGU_Execution_V17".PUMP_1_LINE_FILTER_STATUS = 0) OR
                       ("DB_HGU_Execution_V17".PUMP_1_SUCTION_FILTER_STATUS = 0) OR
                       ("DB_HGU_Execution_V17".PUMP_1_MANUAL_VALVE_STATUS = 0) THEN
                       #Controller_Errors := #Controller_Errors + 1;
                       IF #System_Error_Code = 0 THEN
                           #System_Error_Code := 10 + #i;
                       END_IF; // Safety error codes 11-17
                   END_IF;

               2:
                   IF ("DB_HGU_Execution_V17".PUMP_2_LINE_FILTER_STATUS = 0) OR
                       ("DB_HGU_Execution_V17".PUMP_2_SUCTION_FILTER_STATUS = 0) OR
                       ("DB_HGU_Execution_V17".PUMP_2_MANUAL_VALVE_STATUS = 0) THEN
                       #Controller_Errors := #Controller_Errors + 1;
                       IF #System_Error_Code = 0 THEN
                           #System_Error_Code := 10 + #i;
                       END_IF;
                   END_IF;

               3:
                   IF ("DB_HGU_Execution_V17".PUMP_3_LINE_FILTER_STATUS = 0) OR
                       ("DB_HGU_Execution_V17".PUMP_3_SUCTION_FILTER_STATUS = 0) OR
                       ("DB_HGU_Execution_V17".PUMP_3_MANUAL_VALVE_STATUS = 0) THEN
                       #Controller_Errors := #Controller_Errors + 1;
                       IF #System_Error_Code = 0 THEN
                           #System_Error_Code := 10 + #i;
                       END_IF;
                   END_IF;

               4:
                   IF ("DB_HGU_Execution_V17".PUMP_4_LINE_FILTER_STATUS = 0) OR
                       ("DB_HGU_Execution_V17".PUMP_4_SUCTION_FILTER_STATUS = 0) OR
                       ("DB_HGU_Execution_V17".PUMP_4_MANUAL_VALVE_STATUS = 0) THEN
                       #Controller_Errors := #Controller_Errors + 1;
                       IF #System_Error_Code = 0 THEN
                           #System_Error_Code := 10 + #i;
                       END_IF;
                   END_IF;

               5:
                   IF ("DB_HGU_Execution_V17".PUMP_5_LINE_FILTER_STATUS = 0) OR
                       ("DB_HGU_Execution_V17".PUMP_5_SUCTION_FILTER_STATUS = 0) OR
                       ("DB_HGU_Execution_V17".PUMP_5_MANUAL_VALVE_STATUS = 0) THEN
                       #Controller_Errors := #Controller_Errors + 1;
                       IF #System_Error_Code = 0 THEN
                           #System_Error_Code := 10 + #i;
                       END_IF;
                   END_IF;

               6:
                   IF ("DB_HGU_Execution_V17".PUMP_6_LINE_FILTER_STATUS = 0) OR
                       ("DB_HGU_Execution_V17".PUMP_6_SUCTION_FILTER_STATUS = 0) OR
                       ("DB_HGU_Execution_V17".PUMP_6_MANUAL_VALVE_STATUS = 0) THEN
                       #Controller_Errors := #Controller_Errors + 1;
                       IF #System_Error_Code = 0 THEN
                           #System_Error_Code := 10 + #i;
                       END_IF;
                   END_IF;

               7:
                   IF ("DB_HGU_Execution_V17".PUMP_7_LINE_FILTER_STATUS = 0) OR
                       ("DB_HGU_Execution_V17".PUMP_7_SUCTION_FILTER_STATUS = 0) OR
                       ("DB_HGU_Execution_V17".PUMP_7_MANUAL_VALVE_STATUS = 0) THEN
                       #Controller_Errors := #Controller_Errors + 1;
                       IF #System_Error_Code = 0 THEN
                           #System_Error_Code := 10 + #i;
                       END_IF;
                   END_IF;
           END_CASE;
       END_FOR;

       // Update system safety status
       IF #Controller_Errors > 0 THEN
           "DB_HGU_Execution_V17".SYSTEM_SAFETY_STATUS := 2; // Safety error
       ELSIF #Controller_Errors = 0 THEN
           "DB_HGU_Execution_V17".SYSTEM_SAFETY_STATUS := 1; // All safe
       ELSE
           "DB_HGU_Execution_V17".SYSTEM_SAFETY_STATUS := 0; // Unknown
       END_IF;

       // =============================================================================
       // PRESSURE SETPOINT MANAGEMENT (RISING EDGE + AUTO PROPAGATION)
       // =============================================================================

       // 1. Check for SYSTEM_PRESSURE_SETPOINT rising edge
       #System_Pressure_Changed := ("DB_HGU_Execution_V17".SYSTEM_PRESSURE_SETPOINT <> #Last_System_Pressure_Setpoint);

       // 2. Auto-propagate SYSTEM_PRESSURE_SETPOINT to all pumps when changed
       IF #System_Pressure_Changed THEN
           "DB_HGU_Execution_V17".PUMP_1_PRESSURE_SETPOINT := "DB_HGU_Execution_V17".SYSTEM_PRESSURE_SETPOINT;
           "DB_HGU_Execution_V17".PUMP_2_PRESSURE_SETPOINT := "DB_HGU_Execution_V17".SYSTEM_PRESSURE_SETPOINT;
           "DB_HGU_Execution_V17".PUMP_3_PRESSURE_SETPOINT := "DB_HGU_Execution_V17".SYSTEM_PRESSURE_SETPOINT;
           "DB_HGU_Execution_V17".PUMP_4_PRESSURE_SETPOINT := "DB_HGU_Execution_V17".SYSTEM_PRESSURE_SETPOINT;
           "DB_HGU_Execution_V17".PUMP_5_PRESSURE_SETPOINT := "DB_HGU_Execution_V17".SYSTEM_PRESSURE_SETPOINT;
           "DB_HGU_Execution_V17".PUMP_6_PRESSURE_SETPOINT := "DB_HGU_Execution_V17".SYSTEM_PRESSURE_SETPOINT;
           // NOTE: Motor 7 is separate system - no auto-propagation
       END_IF;

       // 3. Individual pump setpoint check (if any pump > SYSTEM, update SYSTEM and propagate)
       // This creates automatic rising edge for propagation
       FOR #i := 1 TO 6 DO
           CASE #i OF
               1:
                   IF "DB_HGU_Execution_V17".PUMP_1_PRESSURE_SETPOINT > "DB_HGU_Execution_V17".SYSTEM_PRESSURE_SETPOINT THEN
                       "DB_HGU_Execution_V17".SYSTEM_PRESSURE_SETPOINT := "DB_HGU_Execution_V17".PUMP_1_PRESSURE_SETPOINT;
                   END_IF;
               2:
                   IF "DB_HGU_Execution_V17".PUMP_2_PRESSURE_SETPOINT > "DB_HGU_Execution_V17".SYSTEM_PRESSURE_SETPOINT THEN
                       "DB_HGU_Execution_V17".SYSTEM_PRESSURE_SETPOINT := "DB_HGU_Execution_V17".PUMP_2_PRESSURE_SETPOINT;
                   END_IF;
               3:
                   IF "DB_HGU_Execution_V17".PUMP_3_PRESSURE_SETPOINT > "DB_HGU_Execution_V17".SYSTEM_PRESSURE_SETPOINT THEN
                       "DB_HGU_Execution_V17".SYSTEM_PRESSURE_SETPOINT := "DB_HGU_Execution_V17".PUMP_3_PRESSURE_SETPOINT;
                   END_IF;
               4:
                   IF "DB_HGU_Execution_V17".PUMP_4_PRESSURE_SETPOINT > "DB_HGU_Execution_V17".SYSTEM_PRESSURE_SETPOINT THEN
                       "DB_HGU_Execution_V17".SYSTEM_PRESSURE_SETPOINT := "DB_HGU_Execution_V17".PUMP_4_PRESSURE_SETPOINT;
                   END_IF;
               5:
                   IF "DB_HGU_Execution_V17".PUMP_5_PRESSURE_SETPOINT > "DB_HGU_Execution_V17".SYSTEM_PRESSURE_SETPOINT THEN
                       "DB_HGU_Execution_V17".SYSTEM_PRESSURE_SETPOINT := "DB_HGU_Execution_V17".PUMP_5_PRESSURE_SETPOINT;
                   END_IF;
               6:
                   IF "DB_HGU_Execution_V17".PUMP_6_PRESSURE_SETPOINT > "DB_HGU_Execution_V17".SYSTEM_PRESSURE_SETPOINT THEN
                       "DB_HGU_Execution_V17".SYSTEM_PRESSURE_SETPOINT := "DB_HGU_Execution_V17".PUMP_6_PRESSURE_SETPOINT;
                   END_IF;
           END_CASE;
       END_FOR;

       // 4. Update last values for next cycle
       #Last_System_Pressure_Setpoint := "DB_HGU_Execution_V17".SYSTEM_PRESSURE_SETPOINT;

       // =============================================================================
       // SYSTEM STATUS AND MONITORING (FIXED FOR MANIFOLD SYSTEM)
       // =============================================================================

       // Count active motors (separate main system vs Motor 7)
       #Active_Motor_Count := 0;
       #TotalPressure := 0.0;

       // Main system (Motors 1-6): All connected to same manifold
       FOR #i := 1 TO 6 DO
           IF #Motor_Running_Array[#i] THEN
               #Active_Motor_Count := #Active_Motor_Count + 1;

               // For manifold system: use any active pump pressure (they should be same)
               // Take the first active pump pressure as representative
               IF #TotalPressure = 0.0 THEN
                   CASE #i OF
                       1:
                           #TotalPressure := "DB_HGU_Execution_V17".PUMP_1_PRESSURE_ACTUAL;
                       2:
                           #TotalPressure := "DB_HGU_Execution_V17".PUMP_2_PRESSURE_ACTUAL;
                       3:
                           #TotalPressure := "DB_HGU_Execution_V17".PUMP_3_PRESSURE_ACTUAL;
                       4:
                           #TotalPressure := "DB_HGU_Execution_V17".PUMP_4_PRESSURE_ACTUAL;
                       5:
                           #TotalPressure := "DB_HGU_Execution_V17".PUMP_5_PRESSURE_ACTUAL;
                       6:
                           #TotalPressure := "DB_HGU_Execution_V17".PUMP_6_PRESSURE_ACTUAL;
                   END_CASE;
               END_IF;
           END_IF;
       END_FOR;

       // Motor 7 is separate system - count separately but don't add to main pressure
       IF #Motor_Running_Array[7] THEN
           // Motor 7 active pump count separate tracking if needed
           ; // No action for main system pressure calculation
       END_IF;

       // Main system pressure (manifold pressure = any active pump pressure)
       IF #Active_Motor_Count > 0 THEN
           "DB_HGU_Execution_V17".SYSTEM_PRESSURE_AVERAGE := #TotalPressure; // Not average - actual manifold pressure
       ELSE
           "DB_HGU_Execution_V17".SYSTEM_PRESSURE_AVERAGE := 0.0;
       END_IF;

       "DB_HGU_Execution_V17".SYSTEM_ACTIVE_PUMPS := USINT_TO_INT(#Active_Motor_Count);

       // Update outputs
       #Total_System_Flow := #Motor_Selector.Total_Available_Flow;
       #System_Control_Mode := 0; // Default flow control mode

       // =============================================================================
       // SYSTEM STATE MACHINE
       // =============================================================================
       #StateTimer(IN := TRUE,
                   PT := T#2s);

       CASE #SystemState OF
           0: // Initialization
               #SystemReady := FALSE;
               #SystemError := FALSE;
               IF #StateTimer.Q THEN
                   #SystemState := 1;
                   #StateTimer(IN := FALSE,
                               PT := T#2s);
               END_IF;

           1: // Ready
               #SystemReady := TRUE;
               #SystemError := FALSE;
               "DB_HGU_Execution_V17".SYSTEM_STATUS := 1; // Ready
               IF #Active_Motor_Count > 0 THEN
                   #SystemState := 2;
               END_IF;

           2: // Running
               #SystemReady := TRUE;
               #SystemError := FALSE;
               "DB_HGU_Execution_V17".SYSTEM_STATUS := 2; // Running
               IF #Active_Motor_Count = 0 THEN
                   #SystemState := 1;
               END_IF;

               // Check for errors from motor selector
               IF #Motor_Selector.Error_Status THEN
                   #SystemState := 3;
                   #System_Error_Code := #Motor_Selector.Error_Code;
               END_IF;

               // Check for safety errors
               IF #Controller_Errors > 0 THEN
                   #SystemState := 3; // Force error state for safety violations
               END_IF;

           3: // Error
               #SystemReady := FALSE;
               #SystemError := TRUE;
               "DB_HGU_Execution_V17".SYSTEM_STATUS := 3; // Error

               // Error recovery logic
               IF NOT #Motor_Selector.Error_Status AND #Controller_Errors = 0 THEN
                   #SystemState := 1; // Return to ready state
                   #System_Error_Code := 0;
               END_IF;
       END_CASE;

       #SystemStatus := USINT_TO_DINT(#SystemState);

   ELSE
       // =============================================================================
       // SYSTEM DISABLED STATE
       // =============================================================================
       #SystemReady := FALSE;
       #SystemError := FALSE;
       "DB_HGU_Execution_V17".SYSTEM_STATUS := 0; // Disabled
       #SystemState := 0;

       // Disable all controllers
       #Motor_Selector(Enable := FALSE);
       #Dual_Controller_1(Enable := FALSE);
       #Dual_Controller_2(Enable := FALSE);
       #Dual_Controller_3(Enable := FALSE);
       #Dual_Controller_4(Enable := FALSE);
       #Dual_Controller_5(Enable := FALSE);
       #Dual_Controller_6(Enable := FALSE);
       #Dual_Controller_7(Enable := FALSE);

       // Disable all G120C drives
       #G120C_Drive_1(Enable := FALSE);
       #G120C_Drive_2(Enable := FALSE);
       #G120C_Drive_3(Enable := FALSE);
       #G120C_Drive_4(Enable := FALSE);
       #G120C_Drive_5(Enable := FALSE);
       #G120C_Drive_6(Enable := FALSE);

       // Reset all motor outputs
       FOR #i := 1 TO 7 DO
           #Motor_Running_Array[#i] := FALSE;

           CASE #i OF
               1:
                   "DB_HGU_Execution_V17".MOTOR_1_RPM_SETPOINT := 0.0;
                   "DB_HGU_Execution_V17".VALVE_1_CURRENT_SETPOINT := 0.0;
               2:
                   "DB_HGU_Execution_V17".MOTOR_2_RPM_SETPOINT := 0.0;
                   "DB_HGU_Execution_V17".VALVE_2_CURRENT_SETPOINT := 0.0;
               3:
                   "DB_HGU_Execution_V17".MOTOR_3_RPM_SETPOINT := 0.0;
                   "DB_HGU_Execution_V17".VALVE_3_CURRENT_SETPOINT := 0.0;
               4:
                   "DB_HGU_Execution_V17".MOTOR_4_RPM_SETPOINT := 0.0;
                   "DB_HGU_Execution_V17".VALVE_4_CURRENT_SETPOINT := 0.0;
               5:
                   "DB_HGU_Execution_V17".MOTOR_5_RPM_SETPOINT := 0.0;
                   "DB_HGU_Execution_V17".VALVE_5_CURRENT_SETPOINT := 0.0;
               6:
                   "DB_HGU_Execution_V17".MOTOR_6_RPM_SETPOINT := 0.0;
                   "DB_HGU_Execution_V17".VALVE_6_CURRENT_SETPOINT := 0.0;
               7:
                   "DB_HGU_Execution_V17".MOTOR_7_RPM_SETPOINT := 0.0;
                   "DB_HGU_Execution_V17".VALVE_7_CURRENT_SETPOINT := 0.0;
           END_CASE;
       END_FOR;

       #Hour_Update_Timer(IN := FALSE,
                          PT := T#60s);
   END_IF;
END_FUNCTION_BLOCK

